LIN {X 0,Y 319.044,Z 405.7,A -85,B 0,C 180,E1 -15783.168,E2 -15783.168} C_VEL
LIN {X 0,Y 320.819,Z 395.688,A -85,B 0,C 180,E1 -15784.719,E2 -15784.719} C_VEL
LIN {X 0,Y 322.608,Z 384.973,A -85,B 0,C 180,E1 -15786.028,E2 -15786.028} C_VEL
LIN {X 0,Y 324.207,Z 372.814,A -85,B 0,C 180,E1 -15787.203,E2 -15787.203} C_VEL
LIN {X 0,Y 325.391,Z 360.596,A -85,B 0,C 180,E1 -15788.09,E2 -15788.09} C_VEL
LIN {X 0,Y 326.349,Z 347.7,A -85,B 0,C 180,E1 -15788.748,E2 -15788.748} C_VEL
LIN {X 0,Y 326.945,Z 334.043,A -85,B 0,C 180,E1 -15789.178,E2 -15789.178} C_VEL
LIN {X 0,Y 329.007,Z 266.698,A -85,B 0,C 180,E1 -15790.66,E2 -15790.66} C_VEL
LIN {X 0,Y 328.282,Z 264.874,A -85,B 0,C 180,E1 -15790.781,E2 -15790.781} C_VEL
LIN {X 0,Y 325.588,Z 260.147,A -85,B 0,C 180,E1 -15791.184,E2 -15791.184} C_VEL
LIN {X 0,Y 319.666,Z 253.624,A -85,B 0,C 180,E1 -15791.999,E2 -15791.999} C_VEL
LIN {X 0,Y 313.621,Z 247.243,A -85,B 0,C 180,E1 -15792.866,E2 -15792.866} C_VEL
LIN {X 0,Y 310.723,Z 242.716,A -85,B 0,C 180,E1 -15793.339,E2 -15793.339} C_VEL
LIN {X 0,Y 306.192,Z 234.216,A -85,B 0,C 180,E1 -15794.15,E2 -15794.15} C_VEL
LIN {X 0,Y 305.555,Z 231.425,A -85,B 0,C 180,E1 -15795.232,E2 -15795.232} C_VEL
LIN {X 0,Y 305.477,Z 231.432,A -85,B 0,C 180,E1 -15799.393,E2 -15799.393} C_VEL
LIN {X 0,Y 305.486,Z 231.431,A -85,B 0,C 180,E1 -15803.263,E2 -15803.263} C_VEL
LIN {X 0,Y 305.453,Z 231.436,A -85,B 0,C 180,E1 -15806.482,E2 -15806.482} C_VEL
LIN {X 0,Y 305.481,Z 231.426,A -85,B 0,C 180,E1 -15810.95,E2 -15810.95} C_VEL
LIN {X 0,Y 305.557,Z 231.416,A -85,B 0,C 180,E1 -15814.087,E2 -15814.087} C_VEL
LIN {X 0,Y 305.488,Z 231.422,A -85,B 0,C 180,E1 -15818.402,E2 -15818.402} C_VEL
LIN {X 0,Y 305.575,Z 231.42,A -85,B 0,C 180,E1 -15821.217,E2 -15821.217} C_VEL
LIN {X 0,Y 305.632,Z 231.416,A -85,B 0,C 180,E1 -15825.349,E2 -15825.349} C_VEL
LIN {X 0,Y 305.616,Z 231.416,A -85,B 0,C 180,E1 -15829.399,E2 -15829.399} C_VEL
LIN {X 0,Y 305.77,Z 231.385,A -85,B 0,C 180,E1 -15832.074,E2 -15832.074} C_VEL
LIN {X 0,Y 305.664,Z 231.407,A -85,B 0,C 180,E1 -15834.723,E2 -15834.723} C_VEL
LIN {X 0,Y 305.935,Z 231.371,A -85,B 0,C 180,E1 -15838.684,E2 -15838.684} C_VEL
LIN {X 0,Y 305.935,Z 231.362,A -85,B 0,C 180,E1 -15841.317,E2 -15841.317} C_VEL
LIN {X 0,Y 305.65,Z 231.397,A -85,B 0,C 180,E1 -15845.278,E2 -15845.278} C_VEL
LIN {X 0,Y 305.734,Z 231.395,A -85,B 0,C 180,E1 -15847.928,E2 -15847.928} C_VEL
LIN {X 0,Y 305.581,Z 231.414,A -85,B 0,C 180,E1 -15851.946,E2 -15851.946} C_VEL
LIN {X 0,Y 305.592,Z 231.407,A -85,B 0,C 180,E1 -15855.013,E2 -15855.013} C_VEL
LIN {X 0,Y 305.497,Z 231.421,A -85,B 0,C 180,E1 -15858.789,E2 -15858.789} C_VEL
LIN {X 0,Y 305.475,Z 231.425,A -85,B 0,C 180,E1 -15863.041,E2 -15863.041} C_VEL
LIN {X 0,Y 305.456,Z 231.435,A -85,B 0,C 180,E1 -15866.197,E2 -15866.197} C_VEL
LIN {X 0,Y 305.435,Z 231.44,A -85,B 0,C 180,E1 -15869.034,E2 -15869.034} C_VEL
LIN {X 0,Y 305.423,Z 231.436,A -85,B 0,C 180,E1 -15871.955,E2 -15871.955} C_VEL
LIN {X 0,Y 305.45,Z 231.434,A -85,B 0,C 180,E1 -15875.115,E2 -15875.115} C_VEL
LIN {X 0,Y 305.426,Z 231.439,A -85,B 0,C 180,E1 -15878.526,E2 -15878.526} C_VEL
LIN {X 0,Y 305.42,Z 231.421,A -85,B 0,C 180,E1 -15881.861,E2 -15881.861} C_VEL
LIN {X 0,Y 305.394,Z 231.441,A -85,B 0,C 180,E1 -15885.513,E2 -15885.513} C_VEL
LIN {X 0,Y 305.407,Z 231.443,A -85,B 0,C 180,E1 -15888.139,E2 -15888.139} C_VEL
LIN {X 0,Y 305.469,Z 231.431,A -85,B 0,C 180,E1 -15892.434,E2 -15892.434} C_VEL
LIN {X 0,Y 305.482,Z 231.57,A -85,B 0,C 180,E1 -15893.005,E2 -15893.005} C_VEL
LIN {X 0,Y 307.845,Z 240.356,A -85,B 0,C 180,E1 -15896.069,E2 -15896.069} C_VEL
LIN {X 0,Y 310.507,Z 251.535,A -85,B 0,C 180,E1 -15899.69,E2 -15899.69} C_VEL
LIN {X 0,Y 311.721,Z 257.855,A -85,B 0,C 180,E1 -15901.611,E2 -15901.611} C_VEL
LIN {X 0,Y 314.185,Z 264.29,A -85,B 0,C 180,E1 -15902.076,E2 -15902.076} C_VEL
LIN {X 0,Y 318.273,Z 283.563,A -85,B 0,C 180,E1 -15903.048,E2 -15903.048} C_VEL
LIN {X 0,Y 321.317,Z 301.733,A -85,B 0,C 180,E1 -15903.846,E2 -15903.846} C_VEL
LIN {X 0,Y 321.763,Z 306.305,A -85,B 0,C 180,E1 -15904.01,E2 -15904.01} C_VEL
LIN {X 0,Y 319.912,Z 367.181,A -85,B 0,C 180,E1 -15905.416,E2 -15905.416} C_VEL
LIN {X 0,Y 318.804,Z 381.015,A -85,B 0,C 180,E1 -15905.975,E2 -15905.975} C_VEL
LIN {X 0,Y 317.356,Z 393.967,A -85,B 0,C 180,E1 -15906.767,E2 -15906.767} C_VEL
LIN {X 0,Y 315.596,Z 405.738,A -85,B 0,C 180,E1 -15907.754,E2 -15907.754} C_VEL
LIN {X 0,Y 313.641,Z 417.083,A -85,B 0,C 180,E1 -15908.99,E2 -15908.99} C_VEL
LIN {X 0,Y 311.742,Z 427.34,A -85,B 0,C 180,E1 -15910.406,E2 -15910.406} C_VEL
LIN {X 0,Y 310.065,Z 435.756,A -85,B 0,C 180,E1 -15911.84,E2 -15911.84} C_VEL
LIN {X 0,Y 308.386,Z 443.923,A -85,B 0,C 180,E1 -15913.539,E2 -15913.539} C_VEL
LIN {X 0,Y 306.93,Z 451.203,A -85,B 0,C 180,E1 -15915.411,E2 -15915.411} C_VEL
LIN {X 0,Y 305.548,Z 457.385,A -85,B 0,C 180,E1 -15917.377,E2 -15917.377} C_VEL
LIN {X 0,Y 304.67,Z 462.324,A -85,B 0,C 180,E1 -15919.364,E2 -15919.364} C_VEL
LIN {X 0,Y 304.061,Z 466.158,A -85,B 0,C 180,E1 -15921.358,E2 -15921.358} C_VEL
LIN {X 0,Y 303.729,Z 468.991,A -85,B 0,C 180,E1 -15923.355,E2 -15923.355} C_VEL
LIN {X 0,Y 303.654,Z 471.313,A -85,B 0,C 180,E1 -15926.017,E2 -15926.017} C_VEL
LIN {X 0,Y 303.655,Z 471.885,A -85,B 0,C 180,E1 -15927.345,E2 -15927.345} C_VEL
LIN {X 0,Y 303.684,Z 472.025,A -85,B 0,C 180,E1 -15928.672,E2 -15928.672} C_VEL
LIN {X 0,Y 303.77,Z 471.772,A -85,B 0,C 180,E1 -15929.998,E2 -15929.998} C_VEL
LIN {X 0,Y 303.724,Z 471.122,A -85,B 0,C 180,E1 -15931.323,E2 -15931.323} C_VEL
LIN {X 0,Y 303.689,Z 470.074,A -85,B 0,C 180,E1 -15932.65,E2 -15932.65} C_VEL
LIN {X 0,Y 303.734,Z 468.569,A -85,B 0,C 180,E1 -15933.978,E2 -15933.978} C_VEL
LIN {X 0,Y 303.73,Z 465.919,A -85,B 0,C 180,E1 -15935.741,E2 -15935.741} C_VEL
LIN {X 0,Y 303.922,Z 461.34,A -85,B 0,C 180,E1 -15937.972,E2 -15937.972} C_VEL
LIN {X 0,Y 304.388,Z 454.961,A -85,B 0,C 180,E1 -15940.305,E2 -15940.305} C_VEL
LIN {X 0,Y 305.056,Z 448,A -85,B 0,C 180,E1 -15942.301,E2 -15942.301} C_VEL
LIN {X 0,Y 305.854,Z 440.881,A -85,B 0,C 180,E1 -15943.958,E2 -15943.958} C_VEL
LIN {X 0,Y 306.85,Z 432.799,A -85,B 0,C 180,E1 -15945.515,E2 -15945.515} C_VEL
LIN {X 0,Y 307.982,Z 422.94,A -85,B 0,C 180,E1 -15947.065,E2 -15947.065} C_VEL
LIN {X 0,Y 309.065,Z 412.504,A -85,B 0,C 180,E1 -15948.388,E2 -15948.388} C_VEL
LIN {X 0,Y 310.317,Z 401.262,A -85,B 0,C 180,E1 -15949.511,E2 -15949.511} C_VEL
LIN {X 0,Y 311.486,Z 388.684,A -85,B 0,C 180,E1 -15950.466,E2 -15950.466} C_VEL
LIN {X 0,Y 312.401,Z 375.211,A -85,B 0,C 180,E1 -15951.179,E2 -15951.179} C_VEL
LIN {X 0,Y 312.939,Z 361.946,A -85,B 0,C 180,E1 -15951.616,E2 -15951.616} C_VEL
LIN {X 0,Y 314.065,Z 301.944,A -85,B 0,C 180,E1 -15952.983,E2 -15952.983} C_VEL
LIN {X 0,Y 308.541,Z 258.947,A -85,B 0,C 180,E1 -15954.397,E2 -15954.397} C_VEL
LIN {X 0,Y 309.359,Z 251.47,A -85,B 0,C 180,E1 -15956.29,E2 -15956.29} C_VEL
LIN {X 0,Y 308.187,Z 244.192,A -85,B 0,C 180,E1 -15958.278,E2 -15958.278} C_VEL
LIN {X 0,Y 305.47,Z 231.437,A -85,B 0,C 180,E1 -15961.943,E2 -15961.943} C_VEL
LIN {X 0,Y 305.447,Z 231.437,A -85,B 0,C 180,E1 -15965.109,E2 -15965.109} C_VEL
LIN {X 0,Y 305.449,Z 231.437,A -85,B 0,C 180,E1 -15968.528,E2 -15968.528} C_VEL
LIN {X 0,Y 305.439,Z 231.436,A -85,B 0,C 180,E1 -15972.582,E2 -15972.582} C_VEL
LIN {X 0,Y 305.464,Z 231.434,A -85,B 0,C 180,E1 -15976.351,E2 -15976.351} C_VEL
LIN {X 0,Y 305.458,Z 231.437,A -85,B 0,C 180,E1 -15979.892,E2 -15979.892} C_VEL
LIN {X 0,Y 305.471,Z 231.435,A -85,B 0,C 180,E1 -15983.623,E2 -15983.623} C_VEL
LIN {X 0,Y 305.435,Z 231.435,A -85,B 0,C 180,E1 -15986.479,E2 -15986.479} C_VEL
LIN {X 0,Y 305.462,Z 231.433,A -85,B 0,C 180,E1 -15990.947,E2 -15990.947} C_VEL
LIN {X 0,Y 305.538,Z 231.424,A -85,B 0,C 180,E1 -15994.084,E2 -15994.084} C_VEL
LIN {X 0,Y 305.474,Z 231.431,A -85,B 0,C 180,E1 -15998.4,E2 -15998.4} C_VEL
LIN {X 0,Y 305.555,Z 231.424,A -85,B 0,C 180,E1 -16001.215,E2 -16001.215} C_VEL
LIN {X 0,Y 305.599,Z 231.42,A -85,B 0,C 180,E1 -16005.346,E2 -16005.346} C_VEL
LIN {X 0,Y 305.599,Z 231.419,A -85,B 0,C 180,E1 -16009.398,E2 -16009.398} C_VEL
LIN {X 0,Y 305.774,Z 231.394,A -85,B 0,C 180,E1 -16012.073,E2 -16012.073} C_VEL
LIN {X 0,Y 305.649,Z 231.41,A -85,B 0,C 180,E1 -16014.722,E2 -16014.722} C_VEL
LIN {X 0,Y 305.914,Z 231.37,A -85,B 0,C 180,E1 -16018.683,E2 -16018.683} C_VEL
LIN {X 0,Y 305.913,Z 231.373,A -85,B 0,C 180,E1 -16021.316,E2 -16021.316} C_VEL
LIN {X 0,Y 305.795,Z 231.393,A -85,B 0,C 180,E1 -16026.598,E2 -16026.598} C_VEL
LIN {X 0,Y 305.659,Z 231.409,A -85,B 0,C 180,E1 -16029.262,E2 -16029.262} C_VEL
LIN {X 0,Y 305.544,Z 231.423,A -85,B 0,C 180,E1 -16033.298,E2 -16033.298} C_VEL
LIN {X 0,Y 305.513,Z 231.426,A -85,B 0,C 180,E1 -16036.024,E2 -16036.024} C_VEL
LIN {X 0,Y 305.442,Z 231.433,A -85,B 0,C 180,E1 -16040.19,E2 -16040.19} C_VEL
LIN {X 0,Y 305.463,Z 231.436,A -85,B 0,C 180,E1 -16044.465,E2 -16044.465} C_VEL
LIN {X 0,Y 305.454,Z 231.43,A -85,B 0,C 180,E1 -16047.397,E2 -16047.397} C_VEL
LIN {X 0,Y 305.4,Z 231.435,A -85,B 0,C 180,E1 -16050.415,E2 -16050.415} C_VEL
LIN {X 0,Y 305.432,Z 231.434,A -85,B 0,C 180,E1 -16054.081,E2 -16054.081} C_VEL
LIN {X 0,Y 305.443,Z 231.437,A -85,B 0,C 180,E1 -16056.743,E2 -16056.743} C_VEL
LIN {X 0,Y 305.426,Z 231.436,A -85,B 0,C 180,E1 -16060.603,E2 -16060.603} C_VEL
LIN {X 0,Y 305.399,Z 231.434,A -85,B 0,C 180,E1 -16063.659,E2 -16063.659} C_VEL
LIN {X 0,Y 305.431,Z 231.436,A -85,B 0,C 180,E1 -16067.419,E2 -16067.419} C_VEL
LIN {X 0,Y 305.446,Z 231.433,A -85,B 0,C 180,E1 -16071.6,E2 -16071.6} C_VEL
LIN {X 0,Y 305.443,Z 231.435,A -85,B 0,C 180,E1 -16074.891,E2 -16074.891} C_VEL
LIN {X 0,Y 305.433,Z 231.437,A -85,B 0,C 180,E1 -16078.36,E2 -16078.36} C_VEL
LIN {X 0,Y 305.498,Z 231.427,A -85,B 0,C 180,E1 -16081.117,E2 -16081.117} C_VEL
LIN {X 0,Y 305.558,Z 231.425,A -85,B 0,C 180,E1 -16084.092,E2 -16084.092} C_VEL
LIN {X 0,Y 305.464,Z 231.434,A -85,B 0,C 180,E1 -16088.405,E2 -16088.405} C_VEL
LIN {X 0,Y 305.509,Z 231.428,A -85,B 0,C 180,E1 -16091.217,E2 -16091.217} C_VEL
LIN {X 0,Y 305.62,Z 231.417,A -85,B 0,C 180,E1 -16095.351,E2 -16095.351} C_VEL
LIN {X 0,Y 305.683,Z 231.491,A -85,B 0,C 180,E1 -16100.053,E2 -16100.053} C_VEL
LIN {X 0,Y 306.015,Z 233.11,A -85,B 0,C 180,E1 -16100.55,E2 -16100.55} C_VEL
LIN {X 0,Y 313.091,Z 253.572,A -85,B 0,C 180,E1 -16101.521,E2 -16101.521} C_VEL
LIN {X 0,Y 314.73,Z 260.384,A -85,B 0,C 180,E1 -16101.791,E2 -16101.791} C_VEL
LIN {X 0,Y 314.373,Z 285.11,A -85,B 0,C 180,E1 -16102.361,E2 -16102.361} C_VEL
LIN {X 0,Y 313.059,Z 340.43,A -85,B 0,C 180,E1 -16103.639,E2 -16103.639} C_VEL
LIN {X 0,Y 312.537,Z 353.529,A -85,B 0,C 180,E1 -16104.195,E2 -16104.195} C_VEL
LIN {X 0,Y 311.713,Z 366.216,A -85,B 0,C 180,E1 -16104.991,E2 -16104.991} C_VEL
LIN {X 0,Y 310.841,Z 377.488,A -85,B 0,C 180,E1 -16105.951,E2 -16105.951} C_VEL
LIN {X 0,Y 309.763,Z 388.459,A -85,B 0,C 180,E1 -16107.153,E2 -16107.153} C_VEL
LIN {X 0,Y 308.537,Z 399.618,A -85,B 0,C 180,E1 -16108.697,E2 -16108.697} C_VEL
LIN {X 0,Y 307.373,Z 409.069,A -85,B 0,C 180,E1 -16110.33,E2 -16110.33} C_VEL
LIN {X 0,Y 306.231,Z 418.169,A -85,B 0,C 180,E1 -16112.304,E2 -16112.304} C_VEL
LIN {X 0,Y 305.336,Z 425.506,A -85,B 0,C 180,E1 -16114.292,E2 -16114.292} C_VEL
LIN {X 0,Y 304.812,Z 430.463,A -85,B 0,C 180,E1 -16115.957,E2 -16115.957} C_VEL
LIN {X 0,Y 304.304,Z 435.287,A -85,B 0,C 180,E1 -16117.967,E2 -16117.967} C_VEL
LIN {X 0,Y 303.921,Z 438.991,A -85,B 0,C 180,E1 -16119.989,E2 -16119.989} C_VEL
LIN {X 0,Y 303.705,Z 441.659,A -85,B 0,C 180,E1 -16122.022,E2 -16122.022} C_VEL
LIN {X 0,Y 303.61,Z 443.031,A -85,B 0,C 180,E1 -16123.538,E2 -16123.538} C_VEL
LIN {X 0,Y 303.57,Z 444.114,A -85,B 0,C 180,E1 -16126.131,E2 -16126.131} C_VEL
LIN {X 0,Y 303.831,Z 443.821,A -85,B 0,C 180,E1 -16128.491,E2 -16128.491} C_VEL
LIN {X 0,Y 304.111,Z 442.765,A -85,B 0,C 180,E1 -16130.283,E2 -16130.283} C_VEL
LIN {X 0,Y 304.84,Z 440.106,A -85,B 0,C 180,E1 -16132.753,E2 -16132.753} C_VEL
LIN {X 0,Y 305.807,Z 436.078,A -85,B 0,C 180,E1 -16135.161,E2 -16135.161} C_VEL
LIN {X 0,Y 306.971,Z 431.245,A -85,B 0,C 180,E1 -16137.251,E2 -16137.251} C_VEL
LIN {X 0,Y 308.396,Z 425.023,A -85,B 0,C 180,E1 -16139.338,E2 -16139.338} C_VEL
LIN {X 0,Y 310.196,Z 417.184,A -85,B 0,C 180,E1 -16141.406,E2 -16141.406} C_VEL
LIN {X 0,Y 312.044,Z 408.279,A -85,B 0,C 180,E1 -16143.26,E2 -16143.26} C_VEL
LIN {X 0,Y 314.028,Z 397.812,A -85,B 0,C 180,E1 -16144.993,E2 -16144.993} C_VEL
LIN {X 0,Y 315.886,Z 387.609,A -85,B 0,C 180,E1 -16146.324,E2 -16146.324} C_VEL
LIN {X 0,Y 317.479,Z 376.292,A -85,B 0,C 180,E1 -16147.498,E2 -16147.498} C_VEL
LIN {X 0,Y 318.893,Z 363.613,A -85,B 0,C 180,E1 -16148.504,E2 -16148.504} C_VEL
LIN {X 0,Y 319.966,Z 351.192,A -85,B 0,C 180,E1 -16149.209,E2 -16149.209} C_VEL
LIN {X 0,Y 320.63,Z 338.269,A -85,B 0,C 180,E1 -16149.685,E2 -16149.685} C_VEL
LIN {X 0,Y 322.785,Z 268.396,A -85,B 0,C 180,E1 -16151.271,E2 -16151.271} C_VEL
LIN {X 0,Y 315.4,Z 251.823,A -85,B 0,C 180,E1 -16152.533,E2 -16152.533} C_VEL
LIN {X 0,Y 310.723,Z 242.716,A -85,B 0,C 180,E1 -16153.339,E2 -16153.339} C_VEL
LIN {X 0,Y 308.62,Z 239.663,A -85,B 0,C 180,E1 -16153.686,E2 -16153.686} C_VEL
LIN {X 0,Y 305.921,Z 237.295,A -85,B 0,C 180,E1 -16154.092,E2 -16154.092} C_VEL
LIN {X 0,Y 302.106,Z 234.95,A -85,B 0,C 180,E1 -16154.708,E2 -16154.708} C_VEL
LIN {X 0,Y 299.721,Z 233.736,A -85,B 0,C 180,E1 -16155.281,E2 -16155.281} C_VEL
LIN {X 0,Y 298.523,Z 232.453,A -85,B 0,C 180,E1 -16155.908,E2 -16155.908} C_VEL
LIN {X 0,Y 298.487,Z 232.313,A -85,B 0,C 180,E1 -16155.971,E2 -16155.971} C_VEL
LIN {X 0,Y 298.445,Z 232.311,A -85,B 0,C 180,E1 -16158.897,E2 -16158.897} C_VEL
LIN {X 0,Y 298.455,Z 232.307,A -85,B 0,C 180,E1 -16163.187,E2 -16163.187} C_VEL
LIN {X 0,Y 298.383,Z 232.315,A -85,B 0,C 180,E1 -16167.199,E2 -16167.199} C_VEL
LIN {X 0,Y 298.419,Z 232.307,A -85,B 0,C 180,E1 -16170.615,E2 -16170.615} C_VEL
LIN {X 0,Y 298.47,Z 232.304,A -85,B 0,C 180,E1 -16173.474,E2 -16173.474} C_VEL
LIN {X 0,Y 298.421,Z 232.309,A -85,B 0,C 180,E1 -16176.698,E2 -16176.698} C_VEL
LIN {X 0,Y 298.527,Z 232.297,A -85,B 0,C 180,E1 -16180.756,E2 -16180.756} C_VEL
LIN {X 0,Y 298.577,Z 232.292,A -85,B 0,C 180,E1 -16184.994,E2 -16184.994} C_VEL
LIN {X 0,Y 298.572,Z 232.291,A -85,B 0,C 180,E1 -16189.146,E2 -16189.146} C_VEL
LIN {X 0,Y 298.715,Z 232.264,A -85,B 0,C 180,E1 -16191.885,E2 -16191.885} C_VEL
LIN {X 0,Y 298.635,Z 232.282,A -85,B 0,C 180,E1 -16194.599,E2 -16194.599} C_VEL
LIN {X 0,Y 298.902,Z 232.247,A -85,B 0,C 180,E1 -16198.653,E2 -16198.653} C_VEL
LIN {X 0,Y 298.902,Z 232.238,A -85,B 0,C 180,E1 -16201.348,E2 -16201.348} C_VEL
LIN {X 0,Y 298.62,Z 232.272,A -85,B 0,C 180,E1 -16205.402,E2 -16205.402} C_VEL
LIN {X 0,Y 298.685,Z 232.273,A -85,B 0,C 180,E1 -16208.116,E2 -16208.116} C_VEL
LIN {X 0,Y 298.533,Z 232.292,A -85,B 0,C 180,E1 -16212.233,E2 -16212.233} C_VEL
LIN {X 0,Y 298.531,Z 232.287,A -85,B 0,C 180,E1 -16215.166,E2 -16215.166} C_VEL
LIN {X 0,Y 298.429,Z 232.302,A -85,B 0,C 180,E1 -16219.618,E2 -16219.618} C_VEL
LIN {X 0,Y 298.408,Z 232.305,A -85,B 0,C 180,E1 -16223.602,E2 -16223.602} C_VEL
LIN {X 0,Y 298.396,Z 232.31,A -85,B 0,C 180,E1 -16226.584,E2 -16226.584} C_VEL
LIN {X 0,Y 298.381,Z 232.317,A -85,B 0,C 180,E1 -16229.646,E2 -16229.646} C_VEL
LIN {X 0,Y 298.381,Z 232.318,A -85,B 0,C 180,E1 -16232.802,E2 -16232.802} C_VEL
LIN {X 0,Y 298.395,Z 232.316,A -85,B 0,C 180,E1 -16236.074,E2 -16236.074} C_VEL
LIN {X 0,Y 298.391,Z 232.317,A -85,B 0,C 180,E1 -16239.49,E2 -16239.49} C_VEL
LIN {X 0,Y 298.395,Z 232.305,A -85,B 0,C 180,E1 -16243.105,E2 -16243.105} C_VEL
LIN {X 0,Y 298.366,Z 232.319,A -85,B 0,C 180,E1 -16246.916,E2 -16246.916} C_VEL
LIN {X 0,Y 298.382,Z 232.312,A -85,B 0,C 180,E1 -16251.012,E2 -16251.012} C_VEL
LIN {X 0,Y 298.437,Z 232.426,A -85,B 0,C 180,E1 -16252.193,E2 -16252.193} C_VEL
LIN {X 0,Y 301.241,Z 242.869,A -85,B 0,C 180,E1 -16255.95,E2 -16255.95} C_VEL
LIN {X 0,Y 303.699,Z 253.234,A -85,B 0,C 180,E1 -16259.396,E2 -16259.396} C_VEL
LIN {X 0,Y 304.566,Z 257.611,A -85,B 0,C 180,E1 -16260.723,E2 -16260.723} C_VEL
LIN {X 0,Y 308.328,Z 266.462,A -85,B 0,C 180,E1 -16261.439,E2 -16261.439} C_VEL
LIN {X 0,Y 311.791,Z 282.576,A -85,B 0,C 180,E1 -16262.292,E2 -16262.292} C_VEL
LIN {X 0,Y 315.043,Z 301.543,A -85,B 0,C 180,E1 -16263.167,E2 -16263.167} C_VEL
LIN {X 0,Y 315.638,Z 307.057,A -85,B 0,C 180,E1 -16263.378,E2 -16263.378} C_VEL
LIN {X 0,Y 313.694,Z 367.539,A -85,B 0,C 180,E1 -16264.807,E2 -16264.807} C_VEL
LIN {X 0,Y 312.542,Z 381.147,A -85,B 0,C 180,E1 -16265.373,E2 -16265.373} C_VEL
LIN {X 0,Y 311.033,Z 393.946,A -85,B 0,C 180,E1 -16266.178,E2 -16266.178} C_VEL
LIN {X 0,Y 309.073,Z 406.434,A -85,B 0,C 180,E1 -16267.259,E2 -16267.259} C_VEL
LIN {X 0,Y 307.058,Z 417.592,A -85,B 0,C 180,E1 -16268.518,E2 -16268.518} C_VEL
LIN {X 0,Y 305.067,Z 427.673,A -85,B 0,C 180,E1 -16269.959,E2 -16269.959} C_VEL
LIN {X 0,Y 302.954,Z 437.601,A -85,B 0,C 180,E1 -16271.749,E2 -16271.749} C_VEL
LIN {X 0,Y 301.077,Z 446.377,A -85,B 0,C 180,E1 -16273.732,E2 -16273.732} C_VEL
LIN {X 0,Y 299.522,Z 453.436,A -85,B 0,C 180,E1 -16275.736,E2 -16275.736} C_VEL
LIN {X 0,Y 298.207,Z 459.105,A -85,B 0,C 180,E1 -16277.753,E2 -16277.753} C_VEL
LIN {X 0,Y 297.415,Z 463.603,A -85,B 0,C 180,E1 -16279.79,E2 -16279.79} C_VEL
LIN {X 0,Y 296.871,Z 467.046,A -85,B 0,C 180,E1 -16281.832,E2 -16281.832} C_VEL
LIN {X 0,Y 296.554,Z 470.103,A -85,B 0,C 180,E1 -16284.559,E2 -16284.559} C_VEL
LIN {X 0,Y 296.568,Z 471.046,A -85,B 0,C 180,E1 -16285.921,E2 -16285.921} C_VEL
LIN {X 0,Y 296.578,Z 471.576,A -85,B 0,C 180,E1 -16287.281,E2 -16287.281} C_VEL
LIN {X 0,Y 296.678,Z 471.407,A -85,B 0,C 180,E1 -16289.998,E2 -16289.998} C_VEL
LIN {X 0,Y 296.634,Z 470.733,A -85,B 0,C 180,E1 -16291.355,E2 -16291.355} C_VEL
LIN {X 0,Y 296.613,Z 469.646,A -85,B 0,C 180,E1 -16292.714,E2 -16292.714} C_VEL
LIN {X 0,Y 296.645,Z 468.102,A -85,B 0,C 180,E1 -16294.073,E2 -16294.073} C_VEL
LIN {X 0,Y 296.649,Z 465.699,A -85,B 0,C 180,E1 -16295.707,E2 -16295.707} C_VEL
LIN {X 0,Y 296.779,Z 462.287,A -85,B 0,C 180,E1 -16297.481,E2 -16297.481} C_VEL
LIN {X 0,Y 297.087,Z 457.291,A -85,B 0,C 180,E1 -16299.528,E2 -16299.528} C_VEL
LIN {X 0,Y 297.619,Z 450.987,A -85,B 0,C 180,E1 -16301.576,E2 -16301.576} C_VEL
LIN {X 0,Y 298.613,Z 443.109,A -85,B 0,C 180,E1 -16303.609,E2 -16303.609} C_VEL
LIN {X 0,Y 299.753,Z 433.712,A -85,B 0,C 180,E1 -16305.545,E2 -16305.545} C_VEL
LIN {X 0,Y 300.879,Z 424.081,A -85,B 0,C 180,E1 -16307.147,E2 -16307.147} C_VEL
LIN {X 0,Y 302.115,Z 412.723,A -85,B 0,C 180,E1 -16308.65,E2 -16308.65} C_VEL
LIN {X 0,Y 303.4,Z 401.611,A -85,B 0,C 180,E1 -16309.798,E2 -16309.798} C_VEL
LIN {X 0,Y 304.599,Z 389.286,A -85,B 0,C 180,E1 -16310.773,E2 -16310.773} C_VEL
LIN {X 0,Y 305.532,Z 376.273,A -85,B 0,C 180,E1 -16311.502,E2 -16311.502} C_VEL
LIN {X 0,Y 306.157,Z 362.407,A -85,B 0,C 180,E1 -16311.987,E2 -16311.987} C_VEL
LIN {X 0,Y 307.265,Z 302.142,A -85,B 0,C 180,E1 -16313.397,E2 -16313.397} C_VEL
LIN {X 0,Y 301.713,Z 258.649,A -85,B 0,C 180,E1 -16314.859,E2 -16314.859} C_VEL
LIN {X 0,Y 302.352,Z 252.052,A -85,B 0,C 180,E1 -16316.575,E2 -16316.575} C_VEL
LIN {X 0,Y 300.485,Z 242.026,A -85,B 0,C 180,E1 -16319.412,E2 -16319.412} C_VEL
LIN {X 0,Y 298.406,Z 232.316,A -85,B 0,C 180,E1 -16322.288,E2 -16322.288} C_VEL
LIN {X 0,Y 298.403,Z 232.318,A -85,B 0,C 180,E1 -16326.065,E2 -16326.065} C_VEL
LIN {X 0,Y 298.391,Z 232.317,A -85,B 0,C 180,E1 -16329.482,E2 -16329.482} C_VEL
LIN {X 0,Y 298.379,Z 232.315,A -85,B 0,C 180,E1 -16333.099,E2 -16333.099} C_VEL
LIN {X 0,Y 298.417,Z 232.31,A -85,B 0,C 180,E1 -16336.923,E2 -16336.923} C_VEL
LIN {X 0,Y 298.401,Z 232.312,A -85,B 0,C 180,E1 -16340.512,E2 -16340.512} C_VEL
LIN {X 0,Y 298.403,Z 232.315,A -85,B 0,C 180,E1 -16343.928,E2 -16343.928} C_VEL
LIN {X 0,Y 298.364,Z 232.319,A -85,B 0,C 180,E1 -16347.98,E2 -16347.98} C_VEL
LIN {X 0,Y 298.43,Z 232.31,A -85,B 0,C 180,E1 -16351.9,E2 -16351.9} C_VEL
LIN {X 0,Y 298.455,Z 232.306,A -85,B 0,C 180,E1 -16354.921,E2 -16354.921} C_VEL
LIN {X 0,Y 298.404,Z 232.314,A -85,B 0,C 180,E1 -16357.862,E2 -16357.862} C_VEL
LIN {X 0,Y 298.521,Z 232.297,A -85,B 0,C 180,E1 -16360.755,E2 -16360.755} C_VEL
LIN {X 0,Y 298.549,Z 232.296,A -85,B 0,C 180,E1 -16364.992,E2 -16364.992} C_VEL
LIN {X 0,Y 298.554,Z 232.294,A -85,B 0,C 180,E1 -16369.145,E2 -16369.145} C_VEL
LIN {X 0,Y 298.72,Z 232.273,A -85,B 0,C 180,E1 -16371.884,E2 -16371.884} C_VEL
LIN {X 0,Y 298.62,Z 232.285,A -85,B 0,C 180,E1 -16374.598,E2 -16374.598} C_VEL
LIN {X 0,Y 298.881,Z 232.245,A -85,B 0,C 180,E1 -16378.652,E2 -16378.652} C_VEL
LIN {X 0,Y 298.88,Z 232.248,A -85,B 0,C 180,E1 -16381.347,E2 -16381.347} C_VEL
LIN {X 0,Y 298.74,Z 232.273,A -85,B 0,C 180,E1 -16386.755,E2 -16386.755} C_VEL
LIN {X 0,Y 298.591,Z 232.288,A -85,B 0,C 180,E1 -16389.483,E2 -16389.483} C_VEL
LIN {X 0,Y 298.504,Z 232.299,A -85,B 0,C 180,E1 -16393.617,E2 -16393.617} C_VEL
LIN {X 0,Y 298.447,Z 232.309,A -85,B 0,C 180,E1 -16396.414,E2 -16396.414} C_VEL
LIN {X 0,Y 298.406,Z 232.308,A -85,B 0,C 180,E1 -16399.619,E2 -16399.619} C_VEL
LIN {X 0,Y 298.392,Z 232.313,A -85,B 0,C 180,E1 -16403.603,E2 -16403.603} C_VEL
LIN {X 0,Y 298.424,Z 232.311,A -85,B 0,C 180,E1 -16406.58,E2 -16406.58} C_VEL
LIN {X 0,Y 298.368,Z 232.307,A -85,B 0,C 180,E1 -16409.646,E2 -16409.646} C_VEL
LIN {X 0,Y 298.36,Z 232.316,A -85,B 0,C 180,E1 -16412.804,E2 -16412.804} C_VEL
LIN {X 0,Y 298.415,Z 232.312,A -85,B 0,C 180,E1 -16416.81,E2 -16416.81} C_VEL
LIN {X 0,Y 298.359,Z 232.313,A -85,B 0,C 180,E1 -16421.091,E2 -16421.091} C_VEL
LIN {X 0,Y 298.374,Z 232.308,A -85,B 0,C 180,E1 -16423.107,E2 -16423.107} C_VEL
LIN {X 0,Y 298.38,Z 232.315,A -85,B 0,C 180,E1 -16426.925,E2 -16426.925} C_VEL
LIN {X 0,Y 298.378,Z 232.312,A -85,B 0,C 180,E1 -16431.012,E2 -16431.012} C_VEL
LIN {X 0,Y 298.399,Z 232.312,A -85,B 0,C 180,E1 -16433.934,E2 -16433.934} C_VEL
LIN {X 0,Y 298.377,Z 232.319,A -85,B 0,C 180,E1 -16437.988,E2 -16437.988} C_VEL
LIN {X 0,Y 298.445,Z 232.31,A -85,B 0,C 180,E1 -16441.908,E2 -16441.908} C_VEL
LIN {X 0,Y 298.471,Z 232.304,A -85,B 0,C 180,E1 -16444.928,E2 -16444.928} C_VEL
LIN {X 0,Y 298.413,Z 232.312,A -85,B 0,C 180,E1 -16449.317,E2 -16449.317} C_VEL
LIN {X 0,Y 298.485,Z 232.307,A -85,B 0,C 180,E1 -16452.18,E2 -16452.18} C_VEL
LIN {X 0,Y 298.579,Z 232.293,A -85,B 0,C 180,E1 -16454.998,E2 -16454.998} C_VEL
LIN {X 0,Y 298.605,Z 232.292,A -85,B 0,C 180,E1 -16459.691,E2 -16459.691} C_VEL
LIN {X 0,Y 298.929,Z 233.618,A -85,B 0,C 180,E1 -16460.061,E2 -16460.061} C_VEL
LIN {X 0,Y 306.528,Z 255.371,A -85,B 0,C 180,E1 -16461.136,E2 -16461.136} C_VEL
LIN {X 0,Y 308.176,Z 262.479,A -85,B 0,C 180,E1 -16461.42,E2 -16461.42} C_VEL
LIN {X 0,Y 306.282,Z 340.747,A -85,B 0,C 180,E1 -16463.251,E2 -16463.251} C_VEL
LIN {X 0,Y 305.741,Z 353.817,A -85,B 0,C 180,E1 -16463.817,E2 -16463.817} C_VEL
LIN {X 0,Y 304.892,Z 366.516,A -85,B 0,C 180,E1 -16464.63,E2 -16464.63} C_VEL
LIN {X 0,Y 303.915,Z 378.591,A -85,B 0,C 180,E1 -16465.693,E2 -16465.693} C_VEL
LIN {X 0,Y 302.805,Z 389.648,A -85,B 0,C 180,E1 -16466.952,E2 -16466.952} C_VEL
LIN {X 0,Y 301.541,Z 400.472,A -85,B 0,C 180,E1 -16468.5,E2 -16468.5} C_VEL
LIN {X 0,Y 300.461,Z 408.962,A -85,B 0,C 180,E1 -16470.002,E2 -16470.002} C_VEL
LIN {X 0,Y 299.266,Z 418.149,A -85,B 0,C 180,E1 -16472.021,E2 -16472.021} C_VEL
LIN {X 0,Y 298.335,Z 425.545,A -85,B 0,C 180,E1 -16474.055,E2 -16474.055} C_VEL
LIN {X 0,Y 297.697,Z 431.47,A -85,B 0,C 180,E1 -16476.1,E2 -16476.1} C_VEL
LIN {X 0,Y 297.159,Z 436.156,A -85,B 0,C 180,E1 -16478.16,E2 -16478.16} C_VEL
LIN {X 0,Y 296.798,Z 439.726,A -85,B 0,C 180,E1 -16480.231,E2 -16480.231} C_VEL
LIN {X 0,Y 296.581,Z 442.27,A -85,B 0,C 180,E1 -16482.315,E2 -16482.315} C_VEL
LIN {X 0,Y 296.512,Z 443.423,A -85,B 0,C 180,E1 -16483.712,E2 -16483.712} C_VEL
LIN {X 0,Y 296.44,Z 444.152,A -85,B 0,C 180,E1 -16485.118,E2 -16485.118} C_VEL
LIN {X 0,Y 296.497,Z 444.48,A -85,B 0,C 180,E1 -16486.526,E2 -16486.526} C_VEL
LIN {X 0,Y 296.772,Z 444.148,A -85,B 0,C 180,E1 -16488.692,E2 -16488.692} C_VEL
LIN {X 0,Y 297.146,Z 442.884,A -85,B 0,C 180,E1 -16490.78,E2 -16490.78} C_VEL
LIN {X 0,Y 297.877,Z 440.423,A -85,B 0,C 180,E1 -16493.053,E2 -16493.053} C_VEL
LIN {X 0,Y 298.67,Z 437.241,A -85,B 0,C 180,E1 -16495.059,E2 -16495.059} C_VEL
LIN {X 0,Y 299.914,Z 432.43,A -85,B 0,C 180,E1 -16497.312,E2 -16497.312} C_VEL
LIN {X 0,Y 301.587,Z 425.666,A -85,B 0,C 180,E1 -16499.682,E2 -16499.682} C_VEL
LIN {X 0,Y 303.451,Z 417.893,A -85,B 0,C 180,E1 -16501.795,E2 -16501.795} C_VEL
LIN {X 0,Y 305.227,Z 409.852,A -85,B 0,C 180,E1 -16503.546,E2 -16503.546} C_VEL
LIN {X 0,Y 307.271,Z 399.877,A -85,B 0,C 180,E1 -16505.276,E2 -16505.276} C_VEL
LIN {X 0,Y 309.386,Z 388.762,A -85,B 0,C 180,E1 -16506.796,E2 -16506.796} C_VEL
LIN {X 0,Y 311.048,Z 377.617,A -85,B 0,C 180,E1 -16508.002,E2 -16508.002} C_VEL
LIN {X 0,Y 312.514,Z 365.227,A -85,B 0,C 180,E1 -16509.025,E2 -16509.025} C_VEL
LIN {X 0,Y 313.664,Z 352.5,A -85,B 0,C 180,E1 -16509.788,E2 -16509.788} C_VEL
LIN {X 0,Y 314.372,Z 340.811,A -85,B 0,C 180,E1 -16510.255,E2 -16510.255} C_VEL
LIN {X 0,Y 316.741,Z 270.516,A -85,B 0,C 180,E1 -16511.879,E2 -16511.879} C_VEL
LIN {X 0,Y 310.055,Z 255.508,A -85,B 0,C 180,E1 -16513.068,E2 -16513.068} C_VEL
LIN {X 0,Y 302.281,Z 240.681,A -85,B 0,C 180,E1 -16514.467,E2 -16514.467} C_VEL
LIN {X 0,Y 299.104,Z 234.571,A -85,B 0,C 180,E1 -16515.092,E2 -16515.092} C_VEL
LIN {X 0,Y 298.487,Z 232.313,A -85,B 0,C 180,E1 -16515.971,E2 -16515.971} C_VEL
LIN {X 0,Y 297.915,Z 232.378,A -85,B 0,C 180,E1 -16516.704,E2 -16516.704} C_VEL
LIN {X 0,Y 295.823,Z 232.635,A -85,B 0,C 180,E1 -16518.172,E2 -16518.172} C_VEL
LIN {X 0,Y 292.343,Z 233.199,A -85,B 0,C 180,E1 -16520.405,E2 -16520.405} C_VEL
LIN {X 0,Y 291.418,Z 233.195,A -85,B 0,C 180,E1 -16521.567,E2 -16521.567} C_VEL
LIN {X 0,Y 291.351,Z 233.188,A -85,B 0,C 180,E1 -16521.96,E2 -16521.96} C_VEL
LIN {X 0,Y 291.362,Z 233.184,A -85,B 0,C 180,E1 -16525.093,E2 -16525.093} C_VEL
LIN {X 0,Y 291.359,Z 233.184,A -85,B 0,C 180,E1 -16527.95,E2 -16527.95} C_VEL
LIN {X 0,Y 291.369,Z 233.182,A -85,B 0,C 180,E1 -16531.157,E2 -16531.157} C_VEL
LIN {X 0,Y 291.403,Z 233.178,A -85,B 0,C 180,E1 -16534.271,E2 -16534.271} C_VEL
LIN {X 0,Y 291.368,Z 233.189,A -85,B 0,C 180,E1 -16537.299,E2 -16537.299} C_VEL
LIN {X 0,Y 291.447,Z 233.178,A -85,B 0,C 180,E1 -16540.27,E2 -16540.27} C_VEL
LIN {X 0,Y 291.527,Z 233.169,A -85,B 0,C 180,E1 -16544.634,E2 -16544.634} C_VEL
LIN {X 0,Y 291.517,Z 233.169,A -85,B 0,C 180,E1 -16548.88,E2 -16548.88} C_VEL
LIN {X 0,Y 291.663,Z 233.142,A -85,B 0,C 180,E1 -16551.688,E2 -16551.688} C_VEL
LIN {X 0,Y 291.606,Z 233.158,A -85,B 0,C 180,E1 -16554.468,E2 -16554.468} C_VEL
LIN {X 0,Y 291.869,Z 233.123,A -85,B 0,C 180,E1 -16558.621,E2 -16558.621} C_VEL
LIN {X 0,Y 291.868,Z 233.113,A -85,B 0,C 180,E1 -16561.38,E2 -16561.38} C_VEL
LIN {X 0,Y 291.675,Z 233.141,A -85,B 0,C 180,E1 -16566.92,E2 -16566.92} C_VEL
LIN {X 0,Y 291.553,Z 233.153,A -85,B 0,C 180,E1 -16569.715,E2 -16569.715} C_VEL
LIN {X 0,Y 291.499,Z 233.165,A -85,B 0,C 180,E1 -16573.952,E2 -16573.952} C_VEL
LIN {X 0,Y 291.409,Z 233.184,A -85,B 0,C 180,E1 -16576.823,E2 -16576.823} C_VEL
LIN {X 0,Y 291.379,Z 233.181,A -85,B 0,C 180,E1 -16579.843,E2 -16579.843} C_VEL
LIN {X 0,Y 291.347,Z 233.187,A -85,B 0,C 180,E1 -16584.21,E2 -16584.21} C_VEL
LIN {X 0,Y 291.342,Z 233.186,A -85,B 0,C 180,E1 -16587.28,E2 -16587.28} C_VEL
LIN {X 0,Y 291.305,Z 233.194,A -85,B 0,C 180,E1 -16590.441,E2 -16590.441} C_VEL
LIN {X 0,Y 291.333,Z 233.193,A -85,B 0,C 180,E1 -16593.7,E2 -16593.7} C_VEL
LIN {X 0,Y 291.35,Z 233.188,A -85,B 0,C 180,E1 -16597.25,E2 -16597.25} C_VEL
LIN {X 0,Y 291.321,Z 233.184,A -85,B 0,C 180,E1 -16600.645,E2 -16600.645} C_VEL
LIN {X 0,Y 291.287,Z 233.203,A -85,B 0,C 180,E1 -16604.403,E2 -16604.403} C_VEL
LIN {X 0,Y 291.291,Z 233.203,A -85,B 0,C 180,E1 -16608.413,E2 -16608.413} C_VEL
LIN {X 0,Y 291.375,Z 233.266,A -85,B 0,C 180,E1 -16611.321,E2 -16611.321} C_VEL
LIN {X 0,Y 294.082,Z 243.056,A -85,B 0,C 180,E1 -16615.002,E2 -16615.002} C_VEL
LIN {X 0,Y 296.726,Z 254.326,A -85,B 0,C 180,E1 -16618.883,E2 -16618.883} C_VEL
LIN {X 0,Y 297.315,Z 257.08,A -85,B 0,C 180,E1 -16619.762,E2 -16619.762} C_VEL
LIN {X 0,Y 302.874,Z 269.89,A -85,B 0,C 180,E1 -16620.858,E2 -16620.858} C_VEL
LIN {X 0,Y 306.633,Z 288.345,A -85,B 0,C 180,E1 -16621.84,E2 -16621.84} C_VEL
LIN {X 0,Y 309.503,Z 306.524,A -85,B 0,C 180,E1 -16622.676,E2 -16622.676} C_VEL
LIN {X 0,Y 307.63,Z 366.522,A -85,B 0,C 180,E1 -16624.127,E2 -16624.127} C_VEL
LIN {X 0,Y 306.466,Z 379.782,A -85,B 0,C 180,E1 -16624.67,E2 -16624.67} C_VEL
LIN {X 0,Y 304.903,Z 392.9,A -85,B 0,C 180,E1 -16625.487,E2 -16625.487} C_VEL
LIN {X 0,Y 303.174,Z 403.982,A -85,B 0,C 180,E1 -16626.429,E2 -16626.429} C_VEL
LIN {X 0,Y 300.944,Z 415.535,A -85,B 0,C 180,E1 -16627.698,E2 -16627.698} C_VEL
LIN {X 0,Y 298.881,Z 425.942,A -85,B 0,C 180,E1 -16629.166,E2 -16629.166} C_VEL
LIN {X 0,Y 296.967,Z 434.48,A -85,B 0,C 180,E1 -16630.65,E2 -16630.65} C_VEL
LIN {X 0,Y 295.053,Z 443.131,A -85,B 0,C 180,E1 -16632.507,E2 -16632.507} C_VEL
LIN {X 0,Y 293.173,Z 451.26,A -85,B 0,C 180,E1 -16634.71,E2 -16634.71} C_VEL
LIN {X 0,Y 291.664,Z 457.303,A -85,B 0,C 180,E1 -16636.766,E2 -16636.766} C_VEL
LIN {X 0,Y 290.666,Z 462.114,A -85,B 0,C 180,E1 -16638.845,E2 -16638.845} C_VEL
LIN {X 0,Y 289.993,Z 465.833,A -85,B 0,C 180,E1 -16640.935,E2 -16640.935} C_VEL
LIN {X 0,Y 289.58,Z 468.557,A -85,B 0,C 180,E1 -16643.028,E2 -16643.028} C_VEL
LIN {X 0,Y 289.483,Z 469.924,A -85,B 0,C 180,E1 -16644.5,E2 -16644.5} C_VEL
LIN {X 0,Y 289.465,Z 470.776,A -85,B 0,C 180,E1 -16645.821,E2 -16645.821} C_VEL
LIN {X 0,Y 289.503,Z 471.26,A -85,B 0,C 180,E1 -16647.215,E2 -16647.215} C_VEL
LIN {X 0,Y 289.588,Z 471.042,A -85,B 0,C 180,E1 -16649.998,E2 -16649.998} C_VEL
LIN {X 0,Y 289.548,Z 470.344,A -85,B 0,C 180,E1 -16651.388,E2 -16651.388} C_VEL
LIN {X 0,Y 289.539,Z 469.207,A -85,B 0,C 180,E1 -16652.78,E2 -16652.78} C_VEL
LIN {X 0,Y 289.532,Z 466.345,A -85,B 0,C 180,E1 -16655.108,E2 -16655.108} C_VEL
LIN {X 0,Y 289.705,Z 461.736,A -85,B 0,C 180,E1 -16657.664,E2 -16657.664} C_VEL
LIN {X 0,Y 290.053,Z 456.68,A -85,B 0,C 180,E1 -16659.762,E2 -16659.762} C_VEL
LIN {X 0,Y 290.634,Z 450.306,A -85,B 0,C 180,E1 -16661.858,E2 -16661.858} C_VEL
LIN {X 0,Y 291.628,Z 442.306,A -85,B 0,C 180,E1 -16663.941,E2 -16663.941} C_VEL
LIN {X 0,Y 292.776,Z 433.325,A -85,B 0,C 180,E1 -16665.824,E2 -16665.824} C_VEL
LIN {X 0,Y 294.057,Z 423.048,A -85,B 0,C 180,E1 -16667.558,E2 -16667.558} C_VEL
LIN {X 0,Y 295.171,Z 412.913,A -85,B 0,C 180,E1 -16668.926,E2 -16668.926} C_VEL
LIN {X 0,Y 296.492,Z 401.921,A -85,B 0,C 180,E1 -16670.098,E2 -16670.098} C_VEL
LIN {X 0,Y 297.72,Z 389.766,A -85,B 0,C 180,E1 -16671.095,E2 -16671.095} C_VEL
LIN {X 0,Y 298.645,Z 377.222,A -85,B 0,C 180,E1 -16671.841,E2 -16671.841} C_VEL
LIN {X 0,Y 299.299,Z 364.948,A -85,B 0,C 180,E1 -16672.312,E2 -16672.312} C_VEL
LIN {X 0,Y 300.626,Z 303.521,A -85,B 0,C 180,E1 -16673.784,E2 -16673.784} C_VEL
LIN {X 0,Y 294.869,Z 258.279,A -85,B 0,C 180,E1 -16675.357,E2 -16675.357} C_VEL
LIN {X 0,Y 295.328,Z 252.606,A -85,B 0,C 180,E1 -16676.876,E2 -16676.876} C_VEL
LIN {X 0,Y 293.051,Z 240.865,A -85,B 0,C 180,E1 -16680.303,E2 -16680.303} C_VEL
LIN {X 0,Y 291.357,Z 233.193,A -85,B 0,C 180,E1 -16682.679,E2 -16682.679} C_VEL
LIN {X 0,Y 291.394,Z 233.188,A -85,B 0,C 180,E1 -16687.075,E2 -16687.075} C_VEL
LIN {X 0,Y 291.316,Z 233.196,A -85,B 0,C 180,E1 -16690.638,E2 -16690.638} C_VEL
LIN {X 0,Y 291.294,Z 233.198,A -85,B 0,C 180,E1 -16694.393,E2 -16694.393} C_VEL
LIN {X 0,Y 291.357,Z 233.191,A -85,B 0,C 180,E1 -16698.388,E2 -16698.388} C_VEL
LIN {X 0,Y 291.352,Z 233.191,A -85,B 0,C 180,E1 -16701.158,E2 -16701.158} C_VEL
LIN {X 0,Y 291.34,Z 233.192,A -85,B 0,C 180,E1 -16704.623,E2 -16704.623} C_VEL
LIN {X 0,Y 291.341,Z 233.194,A -85,B 0,C 180,E1 -16707.946,E2 -16707.946} C_VEL
LIN {X 0,Y 291.35,Z 233.191,A -85,B 0,C 180,E1 -16711.154,E2 -16711.154} C_VEL
LIN {X 0,Y 291.385,Z 233.186,A -85,B 0,C 180,E1 -16714.268,E2 -16714.268} C_VEL
LIN {X 0,Y 291.372,Z 233.19,A -85,B 0,C 180,E1 -16717.298,E2 -16717.298} C_VEL
LIN {X 0,Y 291.47,Z 233.175,A -85,B 0,C 180,E1 -16720.271,E2 -16720.271} C_VEL
LIN {X 0,Y 291.48,Z 233.175,A -85,B 0,C 180,E1 -16724.65,E2 -16724.65} C_VEL
LIN {X 0,Y 291.498,Z 233.171,A -85,B 0,C 180,E1 -16728.879,E2 -16728.879} C_VEL
LIN {X 0,Y 291.671,Z 233.152,A -85,B 0,C 180,E1 -16731.687,E2 -16731.687} C_VEL
LIN {X 0,Y 291.591,Z 233.159,A -85,B 0,C 180,E1 -16734.467,E2 -16734.467} C_VEL
LIN {X 0,Y 291.847,Z 233.119,A -85,B 0,C 180,E1 -16738.62,E2 -16738.62} C_VEL
LIN {X 0,Y 291.846,Z 233.123,A -85,B 0,C 180,E1 -16741.379,E2 -16741.379} C_VEL
LIN {X 0,Y 291.688,Z 233.153,A -85,B 0,C 180,E1 -16746.919,E2 -16746.919} C_VEL
LIN {X 0,Y 291.533,Z 233.166,A -85,B 0,C 180,E1 -16749.715,E2 -16749.715} C_VEL
LIN {X 0,Y 291.475,Z 233.174,A -85,B 0,C 180,E1 -16753.952,E2 -16753.952} C_VEL
LIN {X 0,Y 291.392,Z 233.189,A -85,B 0,C 180,E1 -16756.823,E2 -16756.823} C_VEL
LIN {X 0,Y 291.355,Z 233.186,A -85,B 0,C 180,E1 -16759.844,E2 -16759.844} C_VEL
LIN {X 0,Y 291.342,Z 233.193,A -85,B 0,C 180,E1 -16764.21,E2 -16764.21} C_VEL
LIN {X 0,Y 291.367,Z 233.184,A -85,B 0,C 180,E1 -16767.277,E2 -16767.277} C_VEL
LIN {X 0,Y 291.288,Z 233.188,A -85,B 0,C 180,E1 -16770.442,E2 -16770.442} C_VEL
LIN {X 0,Y 291.311,Z 233.19,A -85,B 0,C 180,E1 -16773.702,E2 -16773.702} C_VEL
LIN {X 0,Y 291.345,Z 233.191,A -85,B 0,C 180,E1 -16777.257,E2 -16777.257} C_VEL
LIN {X 0,Y 291.304,Z 233.193,A -85,B 0,C 180,E1 -16780.647,E2 -16780.647} C_VEL
LIN {X 0,Y 291.266,Z 233.198,A -85,B 0,C 180,E1 -16784.406,E2 -16784.406} C_VEL
LIN {X 0,Y 291.303,Z 233.2,A -85,B 0,C 180,E1 -16788.409,E2 -16788.409} C_VEL
LIN {X 0,Y 291.327,Z 233.19,A -85,B 0,C 180,E1 -16791.161,E2 -16791.161} C_VEL
LIN {X 0,Y 291.343,Z 233.193,A -85,B 0,C 180,E1 -16794.63,E2 -16794.63} C_VEL
LIN {X 0,Y 291.354,Z 233.194,A -85,B 0,C 180,E1 -16797.955,E2 -16797.955} C_VEL
LIN {X 0,Y 291.363,Z 233.188,A -85,B 0,C 180,E1 -16801.162,E2 -16801.162} C_VEL
LIN {X 0,Y 291.401,Z 233.187,A -85,B 0,C 180,E1 -16804.276,E2 -16804.276} C_VEL
LIN {X 0,Y 291.362,Z 233.19,A -85,B 0,C 180,E1 -16807.303,E2 -16807.303} C_VEL
LIN {X 0,Y 291.397,Z 233.188,A -85,B 0,C 180,E1 -16810.27,E2 -16810.27} C_VEL
LIN {X 0,Y 291.491,Z 233.177,A -85,B 0,C 180,E1 -16814.669,E2 -16814.669} C_VEL
LIN {X 0,Y 291.571,Z 233.168,A -85,B 0,C 180,E1 -16819.202,E2 -16819.202} C_VEL
LIN {X 0,Y 291.618,Z 233.549,A -85,B 0,C 180,E1 -16819.466,E2 -16819.466} C_VEL
LIN {X 0,Y 292.652,Z 236.348,A -85,B 0,C 180,E1 -16819.67,E2 -16819.67} C_VEL
LIN {X 0,Y 299.992,Z 257.231,A -85,B 0,C 180,E1 -16820.738,E2 -16820.738} C_VEL
LIN {X 0,Y 301.423,Z 262.933,A -85,B 0,C 180,E1 -16820.98,E2 -16820.98} C_VEL
LIN {X 0,Y 299.505,Z 341.307,A -85,B 0,C 180,E1 -16822.86,E2 -16822.86} C_VEL
LIN {X 0,Y 298.913,Z 354.766,A -85,B 0,C 180,E1 -16823.464,E2 -16823.464} C_VEL
LIN {X 0,Y 298.084,Z 366.739,A -85,B 0,C 180,E1 -16824.252,E2 -16824.252} C_VEL
LIN {X 0,Y 297.152,Z 378.046,A -85,B 0,C 180,E1 -16825.254,E2 -16825.254} C_VEL
LIN {X 0,Y 295.995,Z 389.331,A -85,B 0,C 180,E1 -16826.549,E2 -16826.549} C_VEL
LIN {X 0,Y 294.678,Z 400.217,A -85,B 0,C 180,E1 -16828.123,E2 -16828.123} C_VEL
LIN {X 0,Y 293.574,Z 408.802,A -85,B 0,C 180,E1 -16829.659,E2 -16829.659} C_VEL
LIN {X 0,Y 292.481,Z 416.726,A -85,B 0,C 180,E1 -16831.379,E2 -16831.379} C_VEL
LIN {X 0,Y 291.492,Z 424.444,A -85,B 0,C 180,E1 -16833.458,E2 -16833.458} C_VEL
LIN {X 0,Y 290.714,Z 430.646,A -85,B 0,C 180,E1 -16835.551,E2 -16835.551} C_VEL
LIN {X 0,Y 290.194,Z 435.564,A -85,B 0,C 180,E1 -16837.656,E2 -16837.656} C_VEL
LIN {X 0,Y 289.776,Z 439.364,A -85,B 0,C 180,E1 -16839.776,E2 -16839.776} C_VEL
LIN {X 0,Y 289.56,Z 441.331,A -85,B 0,C 180,E1 -16841.198,E2 -16841.198} C_VEL
LIN {X 0,Y 289.425,Z 443.734,A -85,B 0,C 180,E1 -16843.761,E2 -16843.761} C_VEL
LIN {X 0,Y 289.349,Z 444.578,A -85,B 0,C 180,E1 -16845.498,E2 -16845.498} C_VEL
LIN {X 0,Y 289.441,Z 444.841,A -85,B 0,C 180,E1 -16846.941,E2 -16846.941} C_VEL
LIN {X 0,Y 289.733,Z 444.472,A -85,B 0,C 180,E1 -16848.914,E2 -16848.914} C_VEL
LIN {X 0,Y 290.197,Z 443.007,A -85,B 0,C 180,E1 -16851.302,E2 -16851.302} C_VEL
LIN {X 0,Y 290.91,Z 440.756,A -85,B 0,C 180,E1 -16853.361,E2 -16853.361} C_VEL
LIN {X 0,Y 291.879,Z 437.104,A -85,B 0,C 180,E1 -16855.684,E2 -16855.684} C_VEL
LIN {X 0,Y 293.206,Z 432.312,A -85,B 0,C 180,E1 -16857.904,E2 -16857.904} C_VEL
LIN {X 0,Y 294.763,Z 426.307,A -85,B 0,C 180,E1 -16860.046,E2 -16860.046} C_VEL
LIN {X 0,Y 296.717,Z 418.602,A -85,B 0,C 180,E1 -16862.203,E2 -16862.203} C_VEL
LIN {X 0,Y 298.58,Z 410.643,A -85,B 0,C 180,E1 -16863.988,E2 -16863.988} C_VEL
LIN {X 0,Y 300.709,Z 400.81,A -85,B 0,C 180,E1 -16865.752,E2 -16865.752} C_VEL
LIN {X 0,Y 302.674,Z 391.11,A -85,B 0,C 180,E1 -16867.135,E2 -16867.135} C_VEL
LIN {X 0,Y 304.42,Z 380.282,A -85,B 0,C 180,E1 -16868.387,E2 -16868.387} C_VEL
LIN {X 0,Y 306.067,Z 368.085,A -85,B 0,C 180,E1 -16869.476,E2 -16869.476} C_VEL
LIN {X 0,Y 307.328,Z 355.459,A -85,B 0,C 180,E1 -16870.295,E2 -16870.295} C_VEL
LIN {X 0,Y 308.176,Z 342.693,A -85,B 0,C 180,E1 -16870.859,E2 -16870.859} C_VEL
LIN {X 0,Y 309.974,Z 293.201,A -85,B 0,C 180,E1 -16872.046,E2 -16872.046} C_VEL
LIN {X 0,Y 310.56,Z 272.286,A -85,B 0,C 180,E1 -16872.547,E2 -16872.547} C_VEL
LIN {X 0,Y 304.558,Z 258.834,A -85,B 0,C 180,E1 -16873.655,E2 -16873.655} C_VEL
LIN {X 0,Y 297.456,Z 245.139,A -85,B 0,C 180,E1 -16874.982,E2 -16874.982} C_VEL
LIN {X 0,Y 293.243,Z 237.697,A -85,B 0,C 180,E1 -16875.792,E2 -16875.792} C_VEL
LIN {X 0,Y 291.9,Z 234.984,A -85,B 0,C 180,E1 -16876.092,E2 -16876.092} C_VEL
LIN {X 0,Y 291.445,Z 233.182,A -85,B 0,C 180,E1 -16876.88,E2 -16876.88} C_VEL
LIN {X 0,Y 291.369,Z 233.192,A -85,B 0,C 180,E1 -16881.161,E2 -16881.161} C_VEL
LIN {X 0,Y 291.351,Z 233.188,A -85,B 0,C 180,E1 -16881.96,E2 -16881.96} C_VEL
LIN {X 0,Y 290.694,Z 233.273,A -85,B 0,C 180,E1 -16883.113,E2 -16883.113} C_VEL
LIN {X 0,Y 287.825,Z 233.626,A -85,B 0,C 180,E1 -16884.99,E2 -16884.99} C_VEL
LIN {X 0,Y 285.386,Z 233.936,A -85,B 0,C 180,E1 -16886.514,E2 -16886.514} C_VEL
LIN {X 0,Y 284.345,Z 234.059,A -85,B 0,C 180,E1 -16887.696,E2 -16887.696} C_VEL
LIN {X 0,Y 284.264,Z 234.067,A -85,B 0,C 180,E1 -16888.096,E2 -16888.096} C_VEL
LIN {X 0,Y 284.346,Z 234.061,A -85,B 0,C 180,E1 -16890.375,E2 -16890.375} C_VEL
LIN {X 0,Y 284.366,Z 234.061,A -85,B 0,C 180,E1 -16893.586,E2 -16893.586} C_VEL
LIN {X 0,Y 284.353,Z 234.061,A -85,B 0,C 180,E1 -16896.706,E2 -16896.706} C_VEL
LIN {X 0,Y 284.391,Z 234.06,A -85,B 0,C 180,E1 -16901.261,E2 -16901.261} C_VEL
LIN {X 0,Y 284.465,Z 234.049,A -85,B 0,C 180,E1 -16904.47,E2 -16904.47} C_VEL
LIN {X 0,Y 284.469,Z 234.046,A -85,B 0,C 180,E1 -16908.601,E2 -16908.601} C_VEL
LIN {X 0,Y 284.616,Z 234.021,A -85,B 0,C 180,E1 -16911.48,E2 -16911.48} C_VEL
LIN {X 0,Y 284.576,Z 234.033,A -85,B 0,C 180,E1 -16914.331,E2 -16914.331} C_VEL
LIN {X 0,Y 284.835,Z 233.999,A -85,B 0,C 180,E1 -16918.587,E2 -16918.587} C_VEL
LIN {X 0,Y 284.835,Z 233.989,A -85,B 0,C 180,E1 -16921.414,E2 -16921.414} C_VEL
LIN {X 0,Y 284.63,Z 234.02,A -85,B 0,C 180,E1 -16927.092,E2 -16927.092} C_VEL
LIN {X 0,Y 284.499,Z 234.03,A -85,B 0,C 180,E1 -16929.958,E2 -16929.958} C_VEL
LIN {X 0,Y 284.448,Z 234.041,A -85,B 0,C 180,E1 -16934.305,E2 -16934.305} C_VEL
LIN {X 0,Y 284.313,Z 234.059,A -85,B 0,C 180,E1 -16938.745,E2 -16938.745} C_VEL
LIN {X 0,Y 284.315,Z 234.06,A -85,B 0,C 180,E1 -16943.298,E2 -16943.298} C_VEL
LIN {X 0,Y 284.318,Z 234.06,A -85,B 0,C 180,E1 -16947.147,E2 -16947.147} C_VEL
LIN {X 0,Y 284.284,Z 234.071,A -85,B 0,C 180,E1 -16950.092,E2 -16950.092} C_VEL
LIN {X 0,Y 284.276,Z 234.075,A -85,B 0,C 180,E1 -16952.95,E2 -16952.95} C_VEL
LIN {X 0,Y 284.312,Z 234.071,A -85,B 0,C 180,E1 -16956.389,E2 -16956.389} C_VEL
LIN {X 0,Y 284.3,Z 234.066,A -85,B 0,C 180,E1 -16959.996,E2 -16959.996} C_VEL
LIN {X 0,Y 284.243,Z 234.081,A -85,B 0,C 180,E1 -16964.192,E2 -16964.192} C_VEL
LIN {X 0,Y 284.236,Z 234.08,A -85,B 0,C 180,E1 -16968.119,E2 -16968.119} C_VEL
LIN {X 0,Y 284.328,Z 234.197,A -85,B 0,C 180,E1 -16970.427,E2 -16970.427} C_VEL
LIN {X 0,Y 286.845,Z 243.26,A -85,B 0,C 180,E1 -16973.984,E2 -16973.984} C_VEL
LIN {X 0,Y 289.073,Z 252.27,A -85,B 0,C 180,E1 -16977.252,E2 -16977.252} C_VEL
LIN {X 0,Y 290.11,Z 256.803,A -85,B 0,C 180,E1 -16978.752,E2 -16978.752} C_VEL
LIN {X 0,Y 297.172,Z 272.198,A -85,B 0,C 180,E1 -16980.186,E2 -16980.186} C_VEL
LIN {X 0,Y 300.766,Z 290.21,A -85,B 0,C 180,E1 -16981.171,E2 -16981.171} C_VEL
LIN {X 0,Y 303.408,Z 306.943,A -85,B 0,C 180,E1 -16981.968,E2 -16981.968} C_VEL
LIN {X 0,Y 303.209,Z 317.768,A -85,B 0,C 180,E1 -16982.246,E2 -16982.246} C_VEL
LIN {X 0,Y 301.495,Z 366.922,A -85,B 0,C 180,E1 -16983.461,E2 -16983.461} C_VEL
LIN {X 0,Y 300.217,Z 380.78,A -85,B 0,C 180,E1 -16984.058,E2 -16984.058} C_VEL
LIN {X 0,Y 298.662,Z 392.968,A -85,B 0,C 180,E1 -16984.847,E2 -16984.847} C_VEL
LIN {X 0,Y 296.722,Z 404.728,A -85,B 0,C 180,E1 -16985.884,E2 -16985.884} C_VEL
LIN {X 0,Y 294.423,Z 416.076,A -85,B 0,C 180,E1 -16987.176,E2 -16987.176} C_VEL
LIN {X 0,Y 292.275,Z 426.326,A -85,B 0,C 180,E1 -16988.672,E2 -16988.672} C_VEL
LIN {X 0,Y 289.892,Z 436.382,A -85,B 0,C 180,E1 -16990.527,E2 -16990.527} C_VEL
LIN {X 0,Y 287.808,Z 445.15,A -85,B 0,C 180,E1 -16992.568,E2 -16992.568} C_VEL
LIN {X 0,Y 286.048,Z 452.41,A -85,B 0,C 180,E1 -16994.684,E2 -16994.684} C_VEL
LIN {X 0,Y 284.283,Z 458.971,A -85,B 0,C 180,E1 -16997.143,E2 -16997.143} C_VEL
LIN {X 0,Y 283.401,Z 463.346,A -85,B 0,C 180,E1 -16999.28,E2 -16999.28} C_VEL
LIN {X 0,Y 282.782,Z 466.674,A -85,B 0,C 180,E1 -17001.422,E2 -17001.422} C_VEL
LIN {X 0,Y 282.388,Z 469.624,A -85,B 0,C 180,E1 -17004.285,E2 -17004.285} C_VEL
LIN {X 0,Y 282.369,Z 470.497,A -85,B 0,C 180,E1 -17005.716,E2 -17005.716} C_VEL
LIN {X 0,Y 282.428,Z 470.945,A -85,B 0,C 180,E1 -17007.145,E2 -17007.145} C_VEL
LIN {X 0,Y 282.501,Z 470.675,A -85,B 0,C 180,E1 -17009.998,E2 -17009.998} C_VEL
LIN {X 0,Y 282.465,Z 469.944,A -85,B 0,C 180,E1 -17011.423,E2 -17011.423} C_VEL
LIN {X 0,Y 282.466,Z 468.763,A -85,B 0,C 180,E1 -17012.85,E2 -17012.85} C_VEL
LIN {X 0,Y 282.475,Z 467.163,A -85,B 0,C 180,E1 -17014.278,E2 -17014.278} C_VEL
LIN {X 0,Y 282.51,Z 463.921,A -85,B 0,C 180,E1 -17016.424,E2 -17016.424} C_VEL
LIN {X 0,Y 282.747,Z 459.586,A -85,B 0,C 180,E1 -17018.574,E2 -17018.574} C_VEL
LIN {X 0,Y 283.189,Z 454.032,A -85,B 0,C 180,E1 -17020.724,E2 -17020.724} C_VEL
LIN {X 0,Y 283.996,Z 447.085,A -85,B 0,C 180,E1 -17022.865,E2 -17022.865} C_VEL
LIN {X 0,Y 284.859,Z 439.971,A -85,B 0,C 180,E1 -17024.644,E2 -17024.644} C_VEL
LIN {X 0,Y 285.863,Z 431.801,A -85,B 0,C 180,E1 -17026.336,E2 -17026.336} C_VEL
LIN {X 0,Y 287.216,Z 421.937,A -85,B 0,C 180,E1 -17027.99,E2 -17027.99} C_VEL
LIN {X 0,Y 288.465,Z 411.645,A -85,B 0,C 180,E1 -17029.383,E2 -17029.383} C_VEL
LIN {X 0,Y 289.774,Z 400.413,A -85,B 0,C 180,E1 -17030.585,E2 -17030.585} C_VEL
LIN {X 0,Y 290.961,Z 389.076,A -85,B 0,C 180,E1 -17031.517,E2 -17031.517} C_VEL
LIN {X 0,Y 291.946,Z 376.319,A -85,B 0,C 180,E1 -17032.276,E2 -17032.276} C_VEL
LIN {X 0,Y 292.621,Z 362.77,A -85,B 0,C 180,E1 -17032.784,E2 -17032.784} C_VEL
LIN {X 0,Y 293.833,Z 303.65,A -85,B 0,C 180,E1 -17034.232,E2 -17034.232} C_VEL
LIN {X 0,Y 288.02,Z 258.035,A -85,B 0,C 180,E1 -17035.846,E2 -17035.846} C_VEL
LIN {X 0,Y 288.397,Z 254.566,A -85,B 0,C 180,E1 -17036.792,E2 -17036.792} C_VEL
LIN {X 0,Y 287.264,Z 247.97,A -85,B 0,C 180,E1 -17038.735,E2 -17038.735} C_VEL
LIN {X 0,Y 285.001,Z 237.28,A -85,B 0,C 180,E1 -17042.011,E2 -17042.011} C_VEL
LIN {X 0,Y 284.333,Z 234.067,A -85,B 0,C 180,E1 -17043.041,E2 -17043.041} C_VEL
LIN {X 0,Y 284.319,Z 234.072,A -85,B 0,C 180,E1 -17046.381,E2 -17046.381} C_VEL
LIN {X 0,Y 284.289,Z 234.076,A -85,B 0,C 180,E1 -17049.99,E2 -17049.99} C_VEL
LIN {X 0,Y 284.246,Z 234.078,A -85,B 0,C 180,E1 -17054.19,E2 -17054.19} C_VEL
LIN {X 0,Y 284.306,Z 234.071,A -85,B 0,C 180,E1 -17058.13,E2 -17058.13} C_VEL
LIN {X 0,Y 284.305,Z 234.072,A -85,B 0,C 180,E1 -17061.829,E2 -17061.829} C_VEL
LIN {X 0,Y 284.283,Z 234.073,A -85,B 0,C 180,E1 -17065.347,E2 -17065.347} C_VEL
LIN {X 0,Y 284.265,Z 234.073,A -85,B 0,C 180,E1 -17068.721,E2 -17068.721} C_VEL
LIN {X 0,Y 284.366,Z 234.06,A -85,B 0,C 180,E1 -17072.823,E2 -17072.823} C_VEL
LIN {X 0,Y 284.345,Z 234.062,A -85,B 0,C 180,E1 -17076.705,E2 -17076.705} C_VEL
LIN {X 0,Y 284.397,Z 234.057,A -85,B 0,C 180,E1 -17079.871,E2 -17079.871} C_VEL
LIN {X 0,Y 284.42,Z 234.054,A -85,B 0,C 180,E1 -17084.484,E2 -17084.484} C_VEL
LIN {X 0,Y 284.45,Z 234.047,A -85,B 0,C 180,E1 -17088.599,E2 -17088.599} C_VEL
LIN {X 0,Y 284.621,Z 234.031,A -85,B 0,C 180,E1 -17091.48,E2 -17091.48} C_VEL
LIN {X 0,Y 284.562,Z 234.035,A -85,B 0,C 180,E1 -17094.33,E2 -17094.33} C_VEL
LIN {X 0,Y 284.813,Z 233.994,A -85,B 0,C 180,E1 -17098.586,E2 -17098.586} C_VEL
LIN {X 0,Y 284.812,Z 233.998,A -85,B 0,C 180,E1 -17101.414,E2 -17101.414} C_VEL
LIN {X 0,Y 284.639,Z 234.03,A -85,B 0,C 180,E1 -17107.091,E2 -17107.091} C_VEL
LIN {X 0,Y 284.478,Z 234.044,A -85,B 0,C 180,E1 -17109.958,E2 -17109.958} C_VEL
LIN {X 0,Y 284.424,Z 234.054,A -85,B 0,C 180,E1 -17114.305,E2 -17114.305} C_VEL
LIN {X 0,Y 284.295,Z 234.07,A -85,B 0,C 180,E1 -17118.745,E2 -17118.745} C_VEL
LIN {X 0,Y 284.295,Z 234.07,A -85,B 0,C 180,E1 -17123.299,E2 -17123.299} C_VEL
LIN {X 0,Y 284.345,Z 234.058,A -85,B 0,C 180,E1 -17127.169,E2 -17127.169} C_VEL
LIN {X 0,Y 284.253,Z 234.062,A -85,B 0,C 180,E1 -17131.279,E2 -17131.279} C_VEL
LIN {X 0,Y 284.311,Z 234.066,A -85,B 0,C 180,E1 -17135.351,E2 -17135.351} C_VEL
LIN {X 0,Y 284.283,Z 234.073,A -85,B 0,C 180,E1 -17138.173,E2 -17138.173} C_VEL
LIN {X 0,Y 284.243,Z 234.071,A -85,B 0,C 180,E1 -17142.128,E2 -17142.128} C_VEL
LIN {X 0,Y 284.232,Z 234.078,A -85,B 0,C 180,E1 -17146.193,E2 -17146.193} C_VEL
LIN {X 0,Y 284.286,Z 234.074,A -85,B 0,C 180,E1 -17150.028,E2 -17150.028} C_VEL
LIN {X 0,Y 284.311,Z 234.064,A -85,B 0,C 180,E1 -17153.618,E2 -17153.618} C_VEL
LIN {X 0,Y 284.291,Z 234.07,A -85,B 0,C 180,E1 -17157.194,E2 -17157.194} C_VEL
LIN {X 0,Y 284.341,Z 234.065,A -85,B 0,C 180,E1 -17160.38,E2 -17160.38} C_VEL
LIN {X 0,Y 284.363,Z 234.063,A -85,B 0,C 180,E1 -17163.591,E2 -17163.591} C_VEL
LIN {X 0,Y 284.322,Z 234.067,A -85,B 0,C 180,E1 -17166.708,E2 -17166.708} C_VEL
LIN {X 0,Y 284.367,Z 234.066,A -85,B 0,C 180,E1 -17169.908,E2 -17169.908} C_VEL
LIN {X 0,Y 284.441,Z 234.056,A -85,B 0,C 180,E1 -17174.496,E2 -17174.496} C_VEL
LIN {X 0,Y 284.507,Z 234.047,A -85,B 0,C 180,E1 -17178.966,E2 -17178.966} C_VEL
LIN {X 0,Y 291.991,Z 254.548,A -85,B 0,C 180,E1 -17180.095,E2 -17180.095} C_VEL
LIN {X 0,Y 294.667,Z 263.566,A -85,B 0,C 180,E1 -17180.524,E2 -17180.524} C_VEL
LIN {X 0,Y 292.815,Z 340.891,A -85,B 0,C 180,E1 -17182.417,E2 -17182.417} C_VEL
LIN {X 0,Y 292.204,Z 354.19,A -85,B 0,C 180,E1 -17183.009,E2 -17183.009} C_VEL
LIN {X 0,Y 291.287,Z 366.962,A -85,B 0,C 180,E1 -17183.857,E2 -17183.857} C_VEL
LIN {X 0,Y 290.237,Z 379.096,A -85,B 0,C 180,E1 -17184.967,E2 -17184.967} C_VEL
LIN {X 0,Y 289.01,Z 390.826,A -85,B 0,C 180,E1 -17186.371,E2 -17186.371} C_VEL
LIN {X 0,Y 287.721,Z 401.022,A -85,B 0,C 180,E1 -17187.903,E2 -17187.903} C_VEL
LIN {X 0,Y 286.427,Z 410.379,A -85,B 0,C 180,E1 -17189.651,E2 -17189.651} C_VEL
LIN {X 0,Y 285.18,Z 419.424,A -85,B 0,C 180,E1 -17191.768,E2 -17191.768} C_VEL
LIN {X 0,Y 284.213,Z 426.713,A -85,B 0,C 180,E1 -17193.901,E2 -17193.901} C_VEL
LIN {X 0,Y 283.602,Z 431.634,A -85,B 0,C 180,E1 -17195.691,E2 -17195.691} C_VEL
LIN {X 0,Y 283.051,Z 436.421,A -85,B 0,C 180,E1 -17197.851,E2 -17197.851} C_VEL
LIN {X 0,Y 282.636,Z 440.09,A -85,B 0,C 180,E1 -17200.026,E2 -17200.026} C_VEL
LIN {X 0,Y 282.45,Z 441.976,A -85,B 0,C 180,E1 -17201.483,E2 -17201.483} C_VEL
LIN {X 0,Y 282.332,Z 444.082,A -85,B 0,C 180,E1 -17203.878,E2 -17203.878} C_VEL
LIN {X 0,Y 282.279,Z 445.002,A -85,B 0,C 180,E1 -17205.896,E2 -17205.896} C_VEL
LIN {X 0,Y 282.416,Z 445.154,A -85,B 0,C 180,E1 -17207.376,E2 -17207.376} C_VEL
LIN {X 0,Y 282.678,Z 444.802,A -85,B 0,C 180,E1 -17209.134,E2 -17209.134} C_VEL
LIN {X 0,Y 283.265,Z 443.101,A -85,B 0,C 180,E1 -17211.849,E2 -17211.849} C_VEL
LIN {X 0,Y 283.936,Z 441.098,A -85,B 0,C 180,E1 -17213.678,E2 -17213.678} C_VEL
LIN {X 0,Y 285.141,Z 436.919,A -85,B 0,C 180,E1 -17216.337,E2 -17216.337} C_VEL
LIN {X 0,Y 286.557,Z 432.048,A -85,B 0,C 180,E1 -17218.571,E2 -17218.571} C_VEL
LIN {X 0,Y 288.27,Z 425.788,A -85,B 0,C 180,E1 -17220.795,E2 -17220.795} C_VEL
LIN {X 0,Y 290.369,Z 417.9,A -85,B 0,C 180,E1 -17222.996,E2 -17222.996} C_VEL
LIN {X 0,Y 292.389,Z 409.687,A -85,B 0,C 180,E1 -17224.81,E2 -17224.81} C_VEL
LIN {X 0,Y 294.626,Z 399.529,A -85,B 0,C 180,E1 -17226.608,E2 -17226.608} C_VEL
LIN {X 0,Y 296.717,Z 389.503,A -85,B 0,C 180,E1 -17228.011,E2 -17228.011} C_VEL
LIN {X 0,Y 298.512,Z 378.6,A -85,B 0,C 180,E1 -17229.239,E2 -17229.239} C_VEL
LIN {X 0,Y 300.131,Z 366.2,A -85,B 0,C 180,E1 -17230.305,E2 -17230.305} C_VEL
LIN {X 0,Y 301.389,Z 353.558,A -85,B 0,C 180,E1 -17231.095,E2 -17231.095} C_VEL
LIN {X 0,Y 302.229,Z 340.528,A -85,B 0,C 180,E1 -17231.628,E2 -17231.628} C_VEL
LIN {X 0,Y 304.625,Z 274.499,A -85,B 0,C 180,E1 -17233.206,E2 -17233.206} C_VEL
LIN {X 0,Y 298.599,Z 261.014,A -85,B 0,C 180,E1 -17234.364,E2 -17234.364} C_VEL
LIN {X 0,Y 289.379,Z 243.471,A -85,B 0,C 180,E1 -17236.178,E2 -17236.178} C_VEL
LIN {X 0,Y 284.688,Z 235.409,A -85,B 0,C 180,E1 -17237.162,E2 -17237.162} C_VEL
LIN {X 0,Y 284.357,Z 234.062,A -85,B 0,C 180,E1 -17237.781,E2 -17237.781} C_VEL
LIN {X 0,Y 284.322,Z 234.065,A -85,B 0,C 180,E1 -17241.964,E2 -17241.964} C_VEL
LIN {X 0,Y 284.3,Z 234.064,A -85,B 0,C 180,E1 -17245.35,E2 -17245.35} C_VEL
LIN {X 0,Y 284.264,Z 234.067,A -85,B 0,C 180,E1 -17248.096,E2 -17248.096} C_VEL
LIN {X 0,Y 283.607,Z 234.154,A -85,B 0,C 180,E1 -17249.279,E2 -17249.279} C_VEL
LIN {X 0,Y 280.767,Z 234.501,A -85,B 0,C 180,E1 -17251.207,E2 -17251.207} C_VEL
LIN {X 0,Y 278.371,Z 234.806,A -85,B 0,C 180,E1 -17252.773,E2 -17252.773} C_VEL
LIN {X 0,Y 277.367,Z 234.928,A -85,B 0,C 180,E1 -17253.986,E2 -17253.986} C_VEL
LIN {X 0,Y 277.298,Z 234.933,A -85,B 0,C 180,E1 -17254.397,E2 -17254.397} C_VEL
LIN {X 0,Y 277.273,Z 234.941,A -85,B 0,C 180,E1 -17257.654,E2 -17257.654} C_VEL
LIN {X 0,Y 277.333,Z 234.937,A -85,B 0,C 180,E1 -17260.766,E2 -17260.766} C_VEL
LIN {X 0,Y 277.413,Z 234.931,A -85,B 0,C 180,E1 -17265.325,E2 -17265.325} C_VEL
LIN {X 0,Y 277.445,Z 234.925,A -85,B 0,C 180,E1 -17269.787,E2 -17269.787} C_VEL
LIN {X 0,Y 277.62,Z 234.893,A -85,B 0,C 180,E1 -17272.729,E2 -17272.729} C_VEL
LIN {X 0,Y 277.801,Z 234.875,A -85,B 0,C 180,E1 -17278.551,E2 -17278.551} C_VEL
LIN {X 0,Y 277.801,Z 234.865,A -85,B 0,C 180,E1 -17281.45,E2 -17281.45} C_VEL
LIN {X 0,Y 277.588,Z 234.898,A -85,B 0,C 180,E1 -17287.273,E2 -17287.273} C_VEL
LIN {X 0,Y 277.44,Z 234.909,A -85,B 0,C 180,E1 -17290.214,E2 -17290.214} C_VEL
LIN {X 0,Y 277.395,Z 234.918,A -85,B 0,C 180,E1 -17294.677,E2 -17294.677} C_VEL
LIN {X 0,Y 277.269,Z 234.936,A -85,B 0,C 180,E1 -17299.24,E2 -17299.24} C_VEL
LIN {X 0,Y 277.27,Z 234.939,A -85,B 0,C 180,E1 -17303.926,E2 -17303.926} C_VEL
LIN {X 0,Y 277.259,Z 234.94,A -85,B 0,C 180,E1 -17307.483,E2 -17307.483} C_VEL
LIN {X 0,Y 277.24,Z 234.945,A -85,B 0,C 180,E1 -17310.474,E2 -17310.474} C_VEL
LIN {X 0,Y 277.231,Z 234.948,A -85,B 0,C 180,E1 -17313.899,E2 -17313.899} C_VEL
LIN {X 0,Y 277.248,Z 234.944,A -85,B 0,C 180,E1 -17317.473,E2 -17317.473} C_VEL
LIN {X 0,Y 277.195,Z 234.936,A -85,B 0,C 180,E1 -17321.24,E2 -17321.24} C_VEL
LIN {X 0,Y 277.191,Z 234.955,A -85,B 0,C 180,E1 -17325.229,E2 -17325.229} C_VEL
LIN {X 0,Y 277.231,Z 235.063,A -85,B 0,C 180,E1 -17329.433,E2 -17329.433} C_VEL
LIN {X 0,Y 280.017,Z 244.824,A -85,B 0,C 180,E1 -17333.433,E2 -17333.433} C_VEL
LIN {X 0,Y 281.955,Z 252.484,A -85,B 0,C 180,E1 -17336.323,E2 -17336.323} C_VEL
LIN {X 0,Y 282.849,Z 256.36,A -85,B 0,C 180,E1 -17337.652,E2 -17337.652} C_VEL
LIN {X 0,Y 290.135,Z 271.788,A -85,B 0,C 180,E1 -17339.211,E2 -17339.211} C_VEL
LIN {X 0,Y 291.882,Z 276.144,A -85,B 0,C 180,E1 -17339.587,E2 -17339.587} C_VEL
LIN {X 0,Y 296.269,Z 299.537,A -85,B 0,C 180,E1 -17340.865,E2 -17340.865} C_VEL
LIN {X 0,Y 297.543,Z 310.385,A -85,B 0,C 180,E1 -17341.341,E2 -17341.341} C_VEL
LIN {X 0,Y 295.461,Z 366.179,A -85,B 0,C 180,E1 -17342.724,E2 -17342.724} C_VEL
LIN {X 0,Y 294.243,Z 379.521,A -85,B 0,C 180,E1 -17343.299,E2 -17343.299} C_VEL
LIN {X 0,Y 292.636,Z 391.979,A -85,B 0,C 180,E1 -17344.1,E2 -17344.1} C_VEL
LIN {X 0,Y 290.589,Z 403.914,A -85,B 0,C 180,E1 -17345.151,E2 -17345.151} C_VEL
LIN {X 0,Y 288.245,Z 415.346,A -85,B 0,C 180,E1 -17346.468,E2 -17346.468} C_VEL
LIN {X 0,Y 285.934,Z 425.669,A -85,B 0,C 180,E1 -17347.986,E2 -17347.986} C_VEL
LIN {X 0,Y 283.628,Z 434.989,A -85,B 0,C 180,E1 -17349.701,E2 -17349.701} C_VEL
LIN {X 0,Y 281.723,Z 442.615,A -85,B 0,C 180,E1 -17351.437,E2 -17351.437} C_VEL
LIN {X 0,Y 279.786,Z 450.223,A -85,B 0,C 180,E1 -17353.584,E2 -17353.584} C_VEL
LIN {X 0,Y 277.834,Z 457.241,A -85,B 0,C 180,E1 -17356.094,E2 -17356.094} C_VEL
LIN {X 0,Y 276.666,Z 461.921,A -85,B 0,C 180,E1 -17358.273,E2 -17358.273} C_VEL
LIN {X 0,Y 275.921,Z 465.52,A -85,B 0,C 180,E1 -17360.468,E2 -17360.468} C_VEL
LIN {X 0,Y 275.454,Z 468.135,A -85,B 0,C 180,E1 -17362.669,E2 -17362.669} C_VEL
LIN {X 0,Y 275.332,Z 469.652,A -85,B 0,C 180,E1 -17364.564,E2 -17364.564} C_VEL
LIN {X 0,Y 275.353,Z 470.63,A -85,B 0,C 180,E1 -17367.072,E2 -17367.072} C_VEL
LIN {X 0,Y 275.351,Z 470.662,A -85,B 0,C 180,E1 -17368.535,E2 -17368.535} C_VEL
LIN {X 0,Y 275.416,Z 470.308,A -85,B 0,C 180,E1 -17369.997,E2 -17369.997} C_VEL
LIN {X 0,Y 275.384,Z 469.53,A -85,B 0,C 180,E1 -17371.46,E2 -17371.46} C_VEL
LIN {X 0,Y 275.394,Z 468.316,A -85,B 0,C 180,E1 -17372.923,E2 -17372.923} C_VEL
LIN {X 0,Y 275.385,Z 465.078,A -85,B 0,C 180,E1 -17375.55,E2 -17375.55} C_VEL
LIN {X 0,Y 275.58,Z 460.609,A -85,B 0,C 180,E1 -17378.06,E2 -17378.06} C_VEL
LIN {X 0,Y 276.056,Z 454.391,A -85,B 0,C 180,E1 -17380.633,E2 -17380.633} C_VEL
LIN {X 0,Y 276.841,Z 447.594,A -85,B 0,C 180,E1 -17382.83,E2 -17382.83} C_VEL
LIN {X 0,Y 277.962,Z 439.142,A -85,B 0,C 180,E1 -17385.016,E2 -17385.016} C_VEL
LIN {X 0,Y 279.186,Z 429.768,A -85,B 0,C 180,E1 -17386.944,E2 -17386.944} C_VEL
LIN {X 0,Y 280.568,Z 419.636,A -85,B 0,C 180,E1 -17388.621,E2 -17388.621} C_VEL
LIN {X 0,Y 281.94,Z 408.931,A -85,B 0,C 180,E1 -17390.04,E2 -17390.04} C_VEL
LIN {X 0,Y 283.353,Z 396.979,A -85,B 0,C 180,E1 -17391.264,E2 -17391.264} C_VEL
LIN {X 0,Y 284.563,Z 384.533,A -85,B 0,C 180,E1 -17392.216,E2 -17392.216} C_VEL
LIN {X 0,Y 285.501,Z 371.736,A -85,B 0,C 180,E1 -17392.903,E2 -17392.903} C_VEL
LIN {X 0,Y 286.012,Z 357.687,A -85,B 0,C 180,E1 -17393.351,E2 -17393.351} C_VEL
LIN {X 0,Y 287.153,Z 304.548,A -85,B 0,C 180,E1 -17394.673,E2 -17394.673} C_VEL
LIN {X 0,Y 281.434,Z 259.259,A -85,B 0,C 180,E1 -17396.312,E2 -17396.312} C_VEL
LIN {X 0,Y 281.241,Z 257.549,A -85,B 0,C 180,E1 -17396.424,E2 -17396.424} C_VEL
LIN {X 0,Y 281.191,Z 253.7,A -85,B 0,C 180,E1 -17397.535,E2 -17397.535} C_VEL
LIN {X 0,Y 278.633,Z 241.199,A -85,B 0,C 180,E1 -17401.409,E2 -17401.409} C_VEL
LIN {X 0,Y 277.275,Z 234.948,A -85,B 0,C 180,E1 -17403.494,E2 -17403.494} C_VEL
LIN {X 0,Y 277.256,Z 234.951,A -85,B 0,C 180,E1 -17407.464,E2 -17407.464} C_VEL
LIN {X 0,Y 277.192,Z 234.956,A -85,B 0,C 180,E1 -17411.232,E2 -17411.232} C_VEL
LIN {X 0,Y 277.21,Z 234.952,A -85,B 0,C 180,E1 -17415.216,E2 -17415.216} C_VEL
LIN {X 0,Y 277.27,Z 234.948,A -85,B 0,C 180,E1 -17419.491,E2 -17419.491} C_VEL
LIN {X 0,Y 277.258,Z 234.946,A -85,B 0,C 180,E1 -17422.529,E2 -17422.529} C_VEL
LIN {X 0,Y 277.22,Z 234.951,A -85,B 0,C 180,E1 -17426.1,E2 -17426.1} C_VEL
LIN {X 0,Y 277.234,Z 234.953,A -85,B 0,C 180,E1 -17429.535,E2 -17429.535} C_VEL
LIN {X 0,Y 277.327,Z 234.937,A -85,B 0,C 180,E1 -17432.86,E2 -17432.86} C_VEL
LIN {X 0,Y 277.311,Z 234.939,A -85,B 0,C 180,E1 -17436.077,E2 -17436.077} C_VEL
LIN {X 0,Y 277.336,Z 234.936,A -85,B 0,C 180,E1 -17440.765,E2 -17440.765} C_VEL
LIN {X 0,Y 277.379,Z 234.936,A -85,B 0,C 180,E1 -17445.322,E2 -17445.322} C_VEL
LIN {X 0,Y 277.469,Z 234.92,A -85,B 0,C 180,E1 -17449.787,E2 -17449.787} C_VEL
LIN {X 0,Y 277.615,Z 234.903,A -85,B 0,C 180,E1 -17452.728,E2 -17452.728} C_VEL
LIN {X 0,Y 277.78,Z 234.869,A -85,B 0,C 180,E1 -17458.55,E2 -17458.55} C_VEL
LIN {X 0,Y 277.779,Z 234.873,A -85,B 0,C 180,E1 -17461.449,E2 -17461.449} C_VEL
LIN {X 0,Y 277.594,Z 234.906,A -85,B 0,C 180,E1 -17467.272,E2 -17467.272} C_VEL
LIN {X 0,Y 277.421,Z 234.924,A -85,B 0,C 180,E1 -17470.214,E2 -17470.214} C_VEL
LIN {X 0,Y 277.371,Z 234.935,A -85,B 0,C 180,E1 -17474.677,E2 -17474.677} C_VEL
LIN {X 0,Y 277.248,Z 234.944,A -85,B 0,C 180,E1 -17479.24,E2 -17479.24} C_VEL
LIN {X 0,Y 277.259,Z 234.946,A -85,B 0,C 180,E1 -17483.926,E2 -17483.926} C_VEL
LIN {X 0,Y 277.275,Z 234.937,A -85,B 0,C 180,E1 -17487.5,E2 -17487.5} C_VEL
LIN {X 0,Y 277.217,Z 234.937,A -85,B 0,C 180,E1 -17490.476,E2 -17490.476} C_VEL
LIN {X 0,Y 277.216,Z 234.946,A -85,B 0,C 180,E1 -17493.899,E2 -17493.899} C_VEL
LIN {X 0,Y 277.238,Z 234.948,A -85,B 0,C 180,E1 -17497.473,E2 -17497.473} C_VEL
LIN {X 0,Y 277.183,Z 234.948,A -85,B 0,C 180,E1 -17501.241,E2 -17501.241} C_VEL
LIN {X 0,Y 277.177,Z 234.952,A -85,B 0,C 180,E1 -17505.231,E2 -17505.231} C_VEL
LIN {X 0,Y 277.201,Z 234.953,A -85,B 0,C 180,E1 -17509.517,E2 -17509.517} C_VEL
LIN {X 0,Y 277.245,Z 234.943,A -85,B 0,C 180,E1 -17512.534,E2 -17512.534} C_VEL
LIN {X 0,Y 277.23,Z 234.954,A -85,B 0,C 180,E1 -17516.108,E2 -17516.108} C_VEL
LIN {X 0,Y 277.247,Z 234.944,A -85,B 0,C 180,E1 -17519.543,E2 -17519.543} C_VEL
LIN {X 0,Y 277.344,Z 234.936,A -85,B 0,C 180,E1 -17522.868,E2 -17522.868} C_VEL
LIN {X 0,Y 277.286,Z 234.946,A -85,B 0,C 180,E1 -17526.081,E2 -17526.081} C_VEL
LIN {X 0,Y 277.303,Z 234.942,A -85,B 0,C 180,E1 -17530.768,E2 -17530.768} C_VEL
LIN {X 0,Y 277.403,Z 234.934,A -85,B 0,C 180,E1 -17535.328,E2 -17535.328} C_VEL
LIN {X 0,Y 277.454,Z 234.927,A -85,B 0,C 180,E1 -17538.424,E2 -17538.424} C_VEL
LIN {X 0,Y 279.163,Z 239.516,A -85,B 0,C 180,E1 -17538.699,E2 -17538.699} C_VEL
LIN {X 0,Y 284.702,Z 254.186,A -85,B 0,C 180,E1 -17539.539,E2 -17539.539} C_VEL
LIN {X 0,Y 288.099,Z 264.99,A -85,B 0,C 180,E1 -17540.083,E2 -17540.083} C_VEL
LIN {X 0,Y 286.001,Z 342.171,A -85,B 0,C 180,E1 -17542.014,E2 -17542.014} C_VEL
LIN {X 0,Y 285.388,Z 355.858,A -85,B 0,C 180,E1 -17542.664,E2 -17542.664} C_VEL
LIN {X 0,Y 284.503,Z 367.178,A -85,B 0,C 180,E1 -17543.443,E2 -17543.443} C_VEL
LIN {X 0,Y 283.504,Z 378.543,A -85,B 0,C 180,E1 -17544.491,E2 -17544.491} C_VEL
LIN {X 0,Y 282.211,Z 390.562,A -85,B 0,C 180,E1 -17545.943,E2 -17545.943} C_VEL
LIN {X 0,Y 280.88,Z 400.762,A -85,B 0,C 180,E1 -17547.493,E2 -17547.493} C_VEL
LIN {X 0,Y 279.552,Z 410.25,A -85,B 0,C 180,E1 -17549.282,E2 -17549.282} C_VEL
LIN {X 0,Y 278.234,Z 419.376,A -85,B 0,C 180,E1 -17551.45,E2 -17551.45} C_VEL
LIN {X 0,Y 277.223,Z 426.73,A -85,B 0,C 180,E1 -17553.636,E2 -17553.636} C_VEL
LIN {X 0,Y 276.487,Z 432.622,A -85,B 0,C 180,E1 -17555.838,E2 -17555.838} C_VEL
LIN {X 0,Y 275.918,Z 437.268,A -85,B 0,C 180,E1 -17558.055,E2 -17558.055} C_VEL
LIN {X 0,Y 275.519,Z 440.809,A -85,B 0,C 180,E1 -17560.287,E2 -17560.287} C_VEL
LIN {X 0,Y 275.323,Z 442.579,A -85,B 0,C 180,E1 -17561.785,E2 -17561.785} C_VEL
LIN {X 0,Y 275.227,Z 444.424,A -85,B 0,C 180,E1 -17563.991,E2 -17563.991} C_VEL
LIN {X 0,Y 275.222,Z 445.384,A -85,B 0,C 180,E1 -17566.315,E2 -17566.315} C_VEL
LIN {X 0,Y 275.384,Z 445.46,A -85,B 0,C 180,E1 -17567.834,E2 -17567.834} C_VEL
LIN {X 0,Y 275.619,Z 445.134,A -85,B 0,C 180,E1 -17569.36,E2 -17569.36} C_VEL
LIN {X 0,Y 275.922,Z 444.389,A -85,B 0,C 180,E1 -17570.892,E2 -17570.892} C_VEL
LIN {X 0,Y 276.367,Z 443.164,A -85,B 0,C 180,E1 -17572.424,E2 -17572.424} C_VEL
LIN {X 0,Y 277.263,Z 440.501,A -85,B 0,C 180,E1 -17574.723,E2 -17574.723} C_VEL
LIN {X 0,Y 278.44,Z 436.721,A -85,B 0,C 180,E1 -17577.022,E2 -17577.022} C_VEL
LIN {X 0,Y 280.002,Z 431.707,A -85,B 0,C 180,E1 -17579.304,E2 -17579.304} C_VEL
LIN {X 0,Y 281.859,Z 425.291,A -85,B 0,C 180,E1 -17581.575,E2 -17581.575} C_VEL
LIN {X 0,Y 284.109,Z 417.135,A -85,B 0,C 180,E1 -17583.819,E2 -17583.819} C_VEL
LIN {X 0,Y 286.447,Z 407.933,A -85,B 0,C 180,E1 -17585.815,E2 -17585.815} C_VEL
LIN {X 0,Y 288.65,Z 398.256,A -85,B 0,C 180,E1 -17587.494,E2 -17587.494} C_VEL
LIN {X 0,Y 290.847,Z 387.786,A -85,B 0,C 180,E1 -17588.921,E2 -17588.921} C_VEL
LIN {X 0,Y 292.593,Z 377.137,A -85,B 0,C 180,E1 -17590.089,E2 -17590.089} C_VEL
LIN {X 0,Y 294.178,Z 365.538,A -85,B 0,C 180,E1 -17591.069,E2 -17591.069} C_VEL
LIN {X 0,Y 295.414,Z 353.028,A -85,B 0,C 180,E1 -17591.848,E2 -17591.848} C_VEL
LIN {X 0,Y 296.225,Z 340.543,A -85,B 0,C 180,E1 -17592.351,E2 -17592.351} C_VEL
LIN {X 0,Y 298.657,Z 276.493,A -85,B 0,C 180,E1 -17593.906,E2 -17593.906} C_VEL
LIN {X 0,Y 292.469,Z 262.861,A -85,B 0,C 180,E1 -17595.146,E2 -17595.146} C_VEL
LIN {X 0,Y 284.486,Z 247.742,A -85,B 0,C 180,E1 -17596.783,E2 -17596.783} C_VEL
LIN {X 0,Y 279.023,Z 238.739,A -85,B 0,C 180,E1 -17597.941,E2 -17597.941} C_VEL
LIN {X 0,Y 277.597,Z 236.296,A -85,B 0,C 180,E1 -17598.257,E2 -17598.257} C_VEL
LIN {X 0,Y 277.382,Z 235.559,A -85,B 0,C 180,E1 -17598.44,E2 -17598.44} C_VEL
LIN {X 0,Y 277.286,Z 234.947,A -85,B 0,C 180,E1 -17598.778,E2 -17598.778} C_VEL
LIN {X 0,Y 277.276,Z 234.941,A -85,B 0,C 180,E1 -17602.533,E2 -17602.533} C_VEL
LIN {X 0,Y 277.238,Z 234.947,A -85,B 0,C 180,E1 -17606.104,E2 -17606.104} C_VEL
LIN {X 0,Y 277.252,Z 234.946,A -85,B 0,C 180,E1 -17609.538,E2 -17609.538} C_VEL
LIN {X 0,Y 277.347,Z 234.933,A -85,B 0,C 180,E1 -17612.863,E2 -17612.863} C_VEL
LIN {X 0,Y 277.298,Z 234.933,A -85,B 0,C 180,E1 -17614.397,E2 -17614.397} C_VEL
LIN {X 0,Y 276.668,Z 235.015,A -85,B 0,C 180,E1 -17615.609,E2 -17615.609} C_VEL
LIN {X 0,Y 273.836,Z 235.372,A -85,B 0,C 180,E1 -17617.584,E2 -17617.584} C_VEL
LIN {X 0,Y 271.405,Z 235.674,A -85,B 0,C 180,E1 -17619.189,E2 -17619.189} C_VEL
LIN {X 0,Y 270.351,Z 235.807,A -85,B 0,C 180,E1 -17620.432,E2 -17620.432} C_VEL
LIN {X 0,Y 270.26,Z 235.812,A -85,B 0,C 180,E1 -17620.854,E2 -17620.854} C_VEL
LIN {X 0,Y 270.382,Z 235.804,A -85,B 0,C 180,E1 -17624.935,E2 -17624.935} C_VEL
LIN {X 0,Y 270.397,Z 235.804,A -85,B 0,C 180,E1 -17629.518,E2 -17629.518} C_VEL
LIN {X 0,Y 270.576,Z 235.769,A -85,B 0,C 180,E1 -17632.538,E2 -17632.538} C_VEL
LIN {X 0,Y 270.768,Z 235.751,A -85,B 0,C 180,E1 -17638.513,E2 -17638.513} C_VEL
LIN {X 0,Y 270.767,Z 235.741,A -85,B 0,C 180,E1 -17641.488,E2 -17641.488} C_VEL
LIN {X 0,Y 270.55,Z 235.777,A -85,B 0,C 180,E1 -17647.463,E2 -17647.463} C_VEL
LIN {X 0,Y 270.374,Z 235.789,A -85,B 0,C 180,E1 -17650.484,E2 -17650.484} C_VEL
LIN {X 0,Y 270.355,Z 235.795,A -85,B 0,C 180,E1 -17655.068,E2 -17655.068} C_VEL
LIN {X 0,Y 270.21,Z 235.817,A -85,B 0,C 180,E1 -17659.763,E2 -17659.763} C_VEL
LIN {X 0,Y 270.214,Z 235.822,A -85,B 0,C 180,E1 -17664.592,E2 -17664.592} C_VEL
LIN {X 0,Y 270.187,Z 235.822,A -85,B 0,C 180,E1 -17667.919,E2 -17667.919} C_VEL
LIN {X 0,Y 270.161,Z 235.825,A -85,B 0,C 180,E1 -17671.352,E2 -17671.352} C_VEL
LIN {X 0,Y 270.187,Z 235.824,A -85,B 0,C 180,E1 -17674.908,E2 -17674.908} C_VEL
LIN {X 0,Y 270.193,Z 235.828,A -85,B 0,C 180,E1 -17678.712,E2 -17678.712} C_VEL
LIN {X 0,Y 270.157,Z 235.822,A -85,B 0,C 180,E1 -17683.249,E2 -17683.249} C_VEL
LIN {X 0,Y 270.148,Z 235.832,A -85,B 0,C 180,E1 -17687.438,E2 -17687.438} C_VEL
LIN {X 0,Y 270.158,Z 235.953,A -85,B 0,C 180,E1 -17688.381,E2 -17688.381} C_VEL
LIN {X 0,Y 272.702,Z 244.538,A -85,B 0,C 180,E1 -17692.097,E2 -17692.097} C_VEL
LIN {X 0,Y 275.088,Z 253.956,A -85,B 0,C 180,E1 -17695.802,E2 -17695.802} C_VEL
LIN {X 0,Y 275.539,Z 255.864,A -85,B 0,C 180,E1 -17696.464,E2 -17696.464} C_VEL
LIN {X 0,Y 282.466,Z 269.97,A -85,B 0,C 180,E1 -17698.026,E2 -17698.026} C_VEL
LIN {X 0,Y 286.328,Z 278.717,A -85,B 0,C 180,E1 -17698.876,E2 -17698.876} C_VEL
LIN {X 0,Y 290.588,Z 302.052,A -85,B 0,C 180,E1 -17700.182,E2 -17700.182} C_VEL
LIN {X 0,Y 291.618,Z 311.28,A -85,B 0,C 180,E1 -17700.596,E2 -17700.596} C_VEL
LIN {X 0,Y 289.453,Z 365.716,A -85,B 0,C 180,E1 -17701.965,E2 -17701.965} C_VEL
LIN {X 0,Y 288.26,Z 379.028,A -85,B 0,C 180,E1 -17702.552,E2 -17702.552} C_VEL
LIN {X 0,Y 286.485,Z 392.067,A -85,B 0,C 180,E1 -17703.403,E2 -17703.403} C_VEL
LIN {X 0,Y 284.206,Z 404.671,A -85,B 0,C 180,E1 -17704.554,E2 -17704.554} C_VEL
LIN {X 0,Y 281.77,Z 415.907,A -85,B 0,C 180,E1 -17705.893,E2 -17705.893} C_VEL
LIN {X 0,Y 279.381,Z 426.06,A -85,B 0,C 180,E1 -17707.441,E2 -17707.441} C_VEL
LIN {X 0,Y 276.977,Z 435.221,A -85,B 0,C 180,E1 -17709.191,E2 -17709.191} C_VEL
LIN {X 0,Y 274.827,Z 443.329,A -85,B 0,C 180,E1 -17711.118,E2 -17711.118} C_VEL
LIN {X 0,Y 272.629,Z 451.399,A -85,B 0,C 180,E1 -17713.526,E2 -17713.526} C_VEL
LIN {X 0,Y 270.94,Z 457.22,A -85,B 0,C 180,E1 -17715.733,E2 -17715.733} C_VEL
LIN {X 0,Y 269.669,Z 461.833,A -85,B 0,C 180,E1 -17717.964,E2 -17717.964} C_VEL
LIN {X 0,Y 268.892,Z 465.373,A -85,B 0,C 180,E1 -17720.217,E2 -17720.217} C_VEL
LIN {X 0,Y 268.378,Z 467.928,A -85,B 0,C 180,E1 -17722.474,E2 -17722.474} C_VEL
LIN {X 0,Y 268.226,Z 469.53,A -85,B 0,C 180,E1 -17724.671,E2 -17724.671} C_VEL
LIN {X 0,Y 268.257,Z 470.314,A -85,B 0,C 180,E1 -17726.994,E2 -17726.994} C_VEL
LIN {X 0,Y 268.273,Z 470.321,A -85,B 0,C 180,E1 -17728.496,E2 -17728.496} C_VEL
LIN {X 0,Y 268.333,Z 469.939,A -85,B 0,C 180,E1 -17729.997,E2 -17729.997} C_VEL
LIN {X 0,Y 268.306,Z 469.11,A -85,B 0,C 180,E1 -17731.498,E2 -17731.498} C_VEL
LIN {X 0,Y 268.323,Z 467.87,A -85,B 0,C 180,E1 -17733,E2 -17733} C_VEL
LIN {X 0,Y 268.288,Z 464.898,A -85,B 0,C 180,E1 -17735.47,E2 -17735.47} C_VEL
LIN {X 0,Y 268.436,Z 461.491,A -85,B 0,C 180,E1 -17737.519,E2 -17737.519} C_VEL
LIN {X 0,Y 268.771,Z 456.631,A -85,B 0,C 180,E1 -17739.782,E2 -17739.782} C_VEL
LIN {X 0,Y 269.361,Z 450.474,A -85,B 0,C 180,E1 -17742.044,E2 -17742.044} C_VEL
LIN {X 0,Y 270.454,Z 442.819,A -85,B 0,C 180,E1 -17744.288,E2 -17744.288} C_VEL
LIN {X 0,Y 271.59,Z 434.971,A -85,B 0,C 180,E1 -17746.147,E2 -17746.147} C_VEL
LIN {X 0,Y 272.679,Z 426.564,A -85,B 0,C 180,E1 -17747.792,E2 -17747.792} C_VEL
LIN {X 0,Y 274.105,Z 415.967,A -85,B 0,C 180,E1 -17749.466,E2 -17749.466} C_VEL
LIN {X 0,Y 275.626,Z 404.37,A -85,B 0,C 180,E1 -17750.91,E2 -17750.91} C_VEL
LIN {X 0,Y 277.02,Z 392.189,A -85,B 0,C 180,E1 -17752.069,E2 -17752.069} C_VEL
LIN {X 0,Y 278.217,Z 378.607,A -85,B 0,C 180,E1 -17752.996,E2 -17752.996} C_VEL
LIN {X 0,Y 279.012,Z 366.032,A -85,B 0,C 180,E1 -17753.565,E2 -17753.565} C_VEL
LIN {X 0,Y 280.459,Z 305.075,A -85,B 0,C 180,E1 -17755.142,E2 -17755.142} C_VEL
LIN {X 0,Y 274.474,Z 257.948,A -85,B 0,C 180,E1 -17756.908,E2 -17756.908} C_VEL
LIN {X 0,Y 274.424,Z 257.341,A -85,B 0,C 180,E1 -17756.951,E2 -17756.951} C_VEL
LIN {X 0,Y 273.47,Z 251.29,A -85,B 0,C 180,E1 -17758.816,E2 -17758.816} C_VEL
LIN {X 0,Y 271.355,Z 241.069,A -85,B 0,C 180,E1 -17762.097,E2 -17762.097} C_VEL
LIN {X 0,Y 270.233,Z 235.827,A -85,B 0,C 180,E1 -17763.875,E2 -17763.875} C_VEL
LIN {X 0,Y 270.213,Z 235.828,A -85,B 0,C 180,E1 -17766.735,E2 -17766.735} C_VEL
LIN {X 0,Y 270.152,Z 235.833,A -85,B 0,C 180,E1 -17771.023,E2 -17771.023} C_VEL
LIN {X 0,Y 270.16,Z 235.831,A -85,B 0,C 180,E1 -17775.381,E2 -17775.381} C_VEL
LIN {X 0,Y 270.221,Z 235.826,A -85,B 0,C 180,E1 -17779.442,E2 -17779.442} C_VEL
LIN {X 0,Y 270.223,Z 235.825,A -85,B 0,C 180,E1 -17783.72,E2 -17783.72} C_VEL
LIN {X 0,Y 270.175,Z 235.827,A -85,B 0,C 180,E1 -17786.888,E2 -17786.888} C_VEL
LIN {X 0,Y 270.2,Z 235.824,A -85,B 0,C 180,E1 -17790.383,E2 -17790.383} C_VEL
LIN {X 0,Y 270.235,Z 235.823,A -85,B 0,C 180,E1 -17793.76,E2 -17793.76} C_VEL
LIN {X 0,Y 270.212,Z 235.824,A -85,B 0,C 180,E1 -17797.036,E2 -17797.036} C_VEL
LIN {X 0,Y 270.293,Z 235.813,A -85,B 0,C 180,E1 -17800.243,E2 -17800.243} C_VEL
LIN {X 0,Y 270.347,Z 235.809,A -85,B 0,C 180,E1 -17804.932,E2 -17804.932} C_VEL
LIN {X 0,Y 270.405,Z 235.801,A -85,B 0,C 180,E1 -17809.517,E2 -17809.517} C_VEL
LIN {X 0,Y 270.574,Z 235.779,A -85,B 0,C 180,E1 -17812.537,E2 -17812.537} C_VEL
LIN {X 0,Y 270.746,Z 235.743,A -85,B 0,C 180,E1 -17818.512,E2 -17818.512} C_VEL
LIN {X 0,Y 270.745,Z 235.747,A -85,B 0,C 180,E1 -17821.487,E2 -17821.487} C_VEL
LIN {X 0,Y 270.551,Z 235.782,A -85,B 0,C 180,E1 -17827.462,E2 -17827.462} C_VEL
LIN {X 0,Y 270.374,Z 235.803,A -85,B 0,C 180,E1 -17830.483,E2 -17830.483} C_VEL
LIN {X 0,Y 270.33,Z 235.812,A -85,B 0,C 180,E1 -17835.068,E2 -17835.068} C_VEL
LIN {X 0,Y 270.188,Z 235.822,A -85,B 0,C 180,E1 -17839.764,E2 -17839.764} C_VEL
LIN {X 0,Y 270.202,Z 235.828,A -85,B 0,C 180,E1 -17844.592,E2 -17844.592} C_VEL
LIN {X 0,Y 270.211,Z 235.817,A -85,B 0,C 180,E1 -17847.915,E2 -17847.915} C_VEL
LIN {X 0,Y 270.143,Z 235.817,A -85,B 0,C 180,E1 -17851.353,E2 -17851.353} C_VEL
LIN {X 0,Y 270.172,Z 235.828,A -85,B 0,C 180,E1 -17854.909,E2 -17854.909} C_VEL
LIN {X 0,Y 270.172,Z 235.829,A -85,B 0,C 180,E1 -17858.714,E2 -17858.714} C_VEL
LIN {X 0,Y 270.14,Z 235.82,A -85,B 0,C 180,E1 -17863.253,E2 -17863.253} C_VEL
LIN {X 0,Y 270.149,Z 235.832,A -85,B 0,C 180,E1 -17867.446,E2 -17867.446} C_VEL
LIN {X 0,Y 270.188,Z 235.822,A -85,B 0,C 180,E1 -17871.378,E2 -17871.378} C_VEL
LIN {X 0,Y 270.184,Z 235.827,A -85,B 0,C 180,E1 -17875.099,E2 -17875.099} C_VEL
LIN {X 0,Y 270.186,Z 235.823,A -85,B 0,C 180,E1 -17879.135,E2 -17879.135} C_VEL
LIN {X 0,Y 270.251,Z 235.823,A -85,B 0,C 180,E1 -17882.151,E2 -17882.151} C_VEL
LIN {X 0,Y 270.226,Z 235.825,A -85,B 0,C 180,E1 -17885.542,E2 -17885.542} C_VEL
LIN {X 0,Y 270.246,Z 235.823,A -85,B 0,C 180,E1 -17890.245,E2 -17890.245} C_VEL
LIN {X 0,Y 270.371,Z 235.809,A -85,B 0,C 180,E1 -17894.938,E2 -17894.938} C_VEL
LIN {X 0,Y 270.383,Z 235.81,A -85,B 0,C 180,E1 -17897.835,E2 -17897.835} C_VEL
LIN {X 0,Y 271.423,Z 238.719,A -85,B 0,C 180,E1 -17898.024,E2 -17898.024} C_VEL
LIN {X 0,Y 276.625,Z 251.533,A -85,B 0,C 180,E1 -17898.824,E2 -17898.824} C_VEL
LIN {X 0,Y 281.454,Z 266.47,A -85,B 0,C 180,E1 -17899.619,E2 -17899.619} C_VEL
LIN {X 0,Y 279.285,Z 342.133,A -85,B 0,C 180,E1 -17901.547,E2 -17901.547} C_VEL
LIN {X 0,Y 278.681,Z 355.19,A -85,B 0,C 180,E1 -17902.167,E2 -17902.167} C_VEL
LIN {X 0,Y 277.732,Z 367.319,A -85,B 0,C 180,E1 -17903.008,E2 -17903.008} C_VEL
LIN {X 0,Y 276.607,Z 379.542,A -85,B 0,C 180,E1 -17904.17,E2 -17904.17} C_VEL
LIN {X 0,Y 275.338,Z 391.093,A -85,B 0,C 180,E1 -17905.611,E2 -17905.611} C_VEL
LIN {X 0,Y 273.937,Z 401.532,A -85,B 0,C 180,E1 -17907.246,E2 -17907.246} C_VEL
LIN {X 0,Y 272.684,Z 410.072,A -85,B 0,C 180,E1 -17908.895,E2 -17908.895} C_VEL
LIN {X 0,Y 271.496,Z 417.94,A -85,B 0,C 180,E1 -17910.744,E2 -17910.744} C_VEL
LIN {X 0,Y 270.364,Z 425.613,A -85,B 0,C 180,E1 -17912.982,E2 -17912.982} C_VEL
LIN {X 0,Y 269.533,Z 431.778,A -85,B 0,C 180,E1 -17915.238,E2 -17915.238} C_VEL
LIN {X 0,Y 268.95,Z 436.67,A -85,B 0,C 180,E1 -17917.509,E2 -17917.509} C_VEL
LIN {X 0,Y 268.498,Z 440.441,A -85,B 0,C 180,E1 -17919.798,E2 -17919.798} C_VEL
LIN {X 0,Y 268.216,Z 443.176,A -85,B 0,C 180,E1 -17922.102,E2 -17922.102} C_VEL
LIN {X 0,Y 268.134,Z 444.769,A -85,B 0,C 180,E1 -17924.119,E2 -17924.119} C_VEL
LIN {X 0,Y 268.175,Z 445.748,A -85,B 0,C 180,E1 -17926.756,E2 -17926.756} C_VEL
LIN {X 0,Y 268.578,Z 445.465,A -85,B 0,C 180,E1 -17929.606,E2 -17929.606} C_VEL
LIN {X 0,Y 268.996,Z 444.52,A -85,B 0,C 180,E1 -17931.456,E2 -17931.456} C_VEL
LIN {X 0,Y 270.034,Z 441.784,A -85,B 0,C 180,E1 -17934.368,E2 -17934.368} C_VEL
LIN {X 0,Y 271.312,Z 437.988,A -85,B 0,C 180,E1 -17936.957,E2 -17936.957} C_VEL
LIN {X 0,Y 272.883,Z 433.246,A -85,B 0,C 180,E1 -17939.297,E2 -17939.297} C_VEL
LIN {X 0,Y 274.763,Z 427.116,A -85,B 0,C 180,E1 -17941.625,E2 -17941.625} C_VEL
LIN {X 0,Y 277.061,Z 419.38,A -85,B 0,C 180,E1 -17943.921,E2 -17943.921} C_VEL
LIN {X 0,Y 279.176,Z 411.642,A -85,B 0,C 180,E1 -17945.757,E2 -17945.757} C_VEL
LIN {X 0,Y 281.399,Z 402.598,A -85,B 0,C 180,E1 -17947.5,E2 -17947.5} C_VEL
LIN {X 0,Y 283.934,Z 391.738,A -85,B 0,C 180,E1 -17949.136,E2 -17949.136} C_VEL
LIN {X 0,Y 286.04,Z 380.351,A -85,B 0,C 180,E1 -17950.504,E2 -17950.504} C_VEL
LIN {X 0,Y 287.789,Z 368.471,A -85,B 0,C 180,E1 -17951.599,E2 -17951.599} C_VEL
LIN {X 0,Y 289.227,Z 355.65,A -85,B 0,C 180,E1 -17952.458,E2 -17952.458} C_VEL
LIN {X 0,Y 290.18,Z 342.569,A -85,B 0,C 180,E1 -17953.048,E2 -17953.048} C_VEL
LIN {X 0,Y 292.641,Z 278.274,A -85,B 0,C 180,E1 -17954.661,E2 -17954.661} C_VEL
LIN {X 0,Y 286.336,Z 264.618,A -85,B 0,C 180,E1 -17955.974,E2 -17955.974} C_VEL
LIN {X 0,Y 279.02,Z 250.926,A -85,B 0,C 180,E1 -17957.543,E2 -17957.543} C_VEL
LIN {X 0,Y 274.437,Z 243.368,A -85,B 0,C 180,E1 -17958.553,E2 -17958.553} C_VEL
LIN {X 0,Y 272.382,Z 240.08,A -85,B 0,C 180,E1 -17959.018,E2 -17959.018} C_VEL
LIN {X 0,Y 270.725,Z 237.61,A -85,B 0,C 180,E1 -17959.395,E2 -17959.395} C_VEL
LIN {X 0,Y 270.306,Z 236.169,A -85,B 0,C 180,E1 -17959.581,E2 -17959.581} C_VEL
LIN {X 0,Y 270.244,Z 235.818,A -85,B 0,C 180,E1 -17959.937,E2 -17959.937} C_VEL
LIN {X 0,Y 270.245,Z 235.823,A -85,B 0,C 180,E1 -17963.722,E2 -17963.722} C_VEL
LIN {X 0,Y 270.193,Z 235.827,A -85,B 0,C 180,E1 -17966.892,E2 -17966.892} C_VEL
LIN {X 0,Y 270.186,Z 235.825,A -85,B 0,C 180,E1 -17970.382,E2 -17970.382} C_VEL
LIN {X 0,Y 270.252,Z 235.816,A -85,B 0,C 180,E1 -17973.763,E2 -17973.763} C_VEL
LIN {X 0,Y 270.221,Z 235.822,A -85,B 0,C 180,E1 -17977.038,E2 -17977.038} C_VEL
LIN {X 0,Y 270.26,Z 235.812,A -85,B 0,C 180,E1 -17980.854,E2 -17980.854} C_VEL
LIN {X 0,Y 269.576,Z 235.899,A -85,B 0,C 180,E1 -17982.098,E2 -17982.098} C_VEL
LIN {X 0,Y 266.717,Z 236.256,A -85,B 0,C 180,E1 -17984.126,E2 -17984.126} C_VEL
LIN {X 0,Y 264.331,Z 236.557,A -85,B 0,C 180,E1 -17985.776,E2 -17985.776} C_VEL
LIN {X 0,Y 263.351,Z 236.671,A -85,B 0,C 180,E1 -17987.054,E2 -17987.054} C_VEL
LIN {X 0,Y 263.294,Z 236.677,A -85,B 0,C 180,E1 -17987.486,E2 -17987.486} C_VEL
LIN {X 0,Y 263.46,Z 236.661,A -85,B 0,C 180,E1 -17990.79,E2 -17990.79} C_VEL
LIN {X 0,Y 263.49,Z 236.661,A -85,B 0,C 180,E1 -17993.876,E2 -17993.876} C_VEL
LIN {X 0,Y 263.733,Z 236.627,A -85,B 0,C 180,E1 -17998.473,E2 -17998.473} C_VEL
LIN {X 0,Y 263.732,Z 236.617,A -85,B 0,C 180,E1 -18001.527,E2 -18001.527} C_VEL
LIN {X 0,Y 263.514,Z 236.654,A -85,B 0,C 180,E1 -18007.664,E2 -18007.664} C_VEL
LIN {X 0,Y 263.321,Z 236.668,A -85,B 0,C 180,E1 -18010.768,E2 -18010.768} C_VEL
LIN {X 0,Y 263.297,Z 236.675,A -85,B 0,C 180,E1 -18015.482,E2 -18015.482} C_VEL
LIN {X 0,Y 263.197,Z 236.694,A -85,B 0,C 180,E1 -18020.312,E2 -18020.312} C_VEL
LIN {X 0,Y 263.157,Z 236.705,A -85,B 0,C 180,E1 -18025.297,E2 -18025.297} C_VEL
LIN {X 0,Y 263.121,Z 236.708,A -85,B 0,C 180,E1 -18028.737,E2 -18028.737} C_VEL
LIN {X 0,Y 263.112,Z 236.708,A -85,B 0,C 180,E1 -18032.292,E2 -18032.292} C_VEL
LIN {X 0,Y 263.15,Z 236.706,A -85,B 0,C 180,E1 -18035.985,E2 -18035.985} C_VEL
LIN {X 0,Y 263.098,Z 236.708,A -85,B 0,C 180,E1 -18039.875,E2 -18039.875} C_VEL
LIN {X 0,Y 263.099,Z 236.713,A -85,B 0,C 180,E1 -18043.99,E2 -18043.99} C_VEL
LIN {X 0,Y 263.119,Z 236.842,A -85,B 0,C 180,E1 -18047.256,E2 -18047.256} C_VEL
LIN {X 0,Y 265.728,Z 245.746,A -85,B 0,C 180,E1 -18051.28,E2 -18051.28} C_VEL
LIN {X 0,Y 268.129,Z 254.746,A -85,B 0,C 180,E1 -18054.994,E2 -18054.994} C_VEL
LIN {X 0,Y 268.275,Z 255.331,A -85,B 0,C 180,E1 -18055.196,E2 -18055.196} C_VEL
LIN {X 0,Y 270.538,Z 259.788,A -85,B 0,C 180,E1 -18055.748,E2 -18055.748} C_VEL
LIN {X 0,Y 277.325,Z 273.48,A -85,B 0,C 180,E1 -18057.335,E2 -18057.335} C_VEL
LIN {X 0,Y 280.916,Z 281.693,A -85,B 0,C 180,E1 -18058.162,E2 -18058.162} C_VEL
LIN {X 0,Y 284.999,Z 305.035,A -85,B 0,C 180,E1 -18059.493,E2 -18059.493} C_VEL
LIN {X 0,Y 285.777,Z 311.178,A -85,B 0,C 180,E1 -18059.792,E2 -18059.792} C_VEL
LIN {X 0,Y 283.502,Z 365.839,A -85,B 0,C 180,E1 -18061.195,E2 -18061.195} C_VEL
LIN {X 0,Y 282.219,Z 379.388,A -85,B 0,C 180,E1 -18061.812,E2 -18061.812} C_VEL
LIN {X 0,Y 280.38,Z 392.203,A -85,B 0,C 180,E1 -18062.676,E2 -18062.676} C_VEL
LIN {X 0,Y 278.147,Z 403.913,A -85,B 0,C 180,E1 -18063.757,E2 -18063.757} C_VEL
LIN {X 0,Y 275.661,Z 415.214,A -85,B 0,C 180,E1 -18065.123,E2 -18065.123} C_VEL
LIN {X 0,Y 273.122,Z 425.437,A -85,B 0,C 180,E1 -18066.694,E2 -18066.694} C_VEL
LIN {X 0,Y 270.358,Z 435.462,A -85,B 0,C 180,E1 -18068.657,E2 -18068.657} C_VEL
LIN {X 0,Y 267.992,Z 443.921,A -85,B 0,C 180,E1 -18070.751,E2 -18070.751} C_VEL
LIN {X 0,Y 265.797,Z 451.448,A -85,B 0,C 180,E1 -18073.09,E2 -18073.09} C_VEL
LIN {X 0,Y 264.047,Z 457.181,A -85,B 0,C 180,E1 -18075.352,E2 -18075.352} C_VEL
LIN {X 0,Y 262.685,Z 461.729,A -85,B 0,C 180,E1 -18077.639,E2 -18077.639} C_VEL
LIN {X 0,Y 262.107,Z 464.143,A -85,B 0,C 180,E1 -18079.18,E2 -18079.18} C_VEL
LIN {X 0,Y 261.667,Z 466.137,A -85,B 0,C 180,E1 -18080.724,E2 -18080.724} C_VEL
LIN {X 0,Y 261.32,Z 467.724,A -85,B 0,C 180,E1 -18082.27,E2 -18082.27} C_VEL
LIN {X 0,Y 261.126,Z 469.402,A -85,B 0,C 180,E1 -18084.768,E2 -18084.768} C_VEL
LIN {X 0,Y 261.164,Z 469.999,A -85,B 0,C 180,E1 -18086.912,E2 -18086.912} C_VEL
LIN {X 0,Y 261.197,Z 469.979,A -85,B 0,C 180,E1 -18088.456,E2 -18088.456} C_VEL
LIN {X 0,Y 261.253,Z 469.553,A -85,B 0,C 180,E1 -18089.997,E2 -18089.997} C_VEL
LIN {X 0,Y 261.229,Z 468.686,A -85,B 0,C 180,E1 -18091.539,E2 -18091.539} C_VEL
LIN {X 0,Y 261.229,Z 467.417,A -85,B 0,C 180,E1 -18093.081,E2 -18093.081} C_VEL
LIN {X 0,Y 261.203,Z 464.672,A -85,B 0,C 180,E1 -18095.413,E2 -18095.413} C_VEL
LIN {X 0,Y 261.358,Z 460.914,A -85,B 0,C 180,E1 -18097.723,E2 -18097.723} C_VEL
LIN {X 0,Y 261.721,Z 455.984,A -85,B 0,C 180,E1 -18100.049,E2 -18100.049} C_VEL
LIN {X 0,Y 262.38,Z 449.753,A -85,B 0,C 180,E1 -18102.37,E2 -18102.37} C_VEL
LIN {X 0,Y 263.506,Z 441.992,A -85,B 0,C 180,E1 -18104.673,E2 -18104.673} C_VEL
LIN {X 0,Y 264.672,Z 434.017,A -85,B 0,C 180,E1 -18106.582,E2 -18106.582} C_VEL
LIN {X 0,Y 266.083,Z 424.265,A -85,B 0,C 180,E1 -18108.474,E2 -18108.474} C_VEL
LIN {X 0,Y 267.482,Z 413.408,A -85,B 0,C 180,E1 -18110.168,E2 -18110.168} C_VEL
LIN {X 0,Y 268.936,Z 402.913,A -85,B 0,C 180,E1 -18111.455,E2 -18111.455} C_VEL
LIN {X 0,Y 270.302,Z 391.414,A -85,B 0,C 180,E1 -18112.546,E2 -18112.546} C_VEL
LIN {X 0,Y 271.55,Z 377.681,A -85,B 0,C 180,E1 -18113.494,E2 -18113.494} C_VEL
LIN {X 0,Y 272.344,Z 364.628,A -85,B 0,C 180,E1 -18114.077,E2 -18114.077} C_VEL
LIN {X 0,Y 273.792,Z 305.788,A -85,B 0,C 180,E1 -18115.627,E2 -18115.627} C_VEL
LIN {X 0,Y 268.03,Z 259.762,A -85,B 0,C 180,E1 -18117.398,E2 -18117.398} C_VEL
LIN {X 0,Y 267.368,Z 256.963,A -85,B 0,C 180,E1 -18117.569,E2 -18117.569} C_VEL
LIN {X 0,Y 264.902,Z 244.639,A -85,B 0,C 180,E1 -18121.579,E2 -18121.579} C_VEL
LIN {X 0,Y 263.189,Z 236.705,A -85,B 0,C 180,E1 -18124.31,E2 -18124.31} C_VEL
LIN {X 0,Y 263.147,Z 236.71,A -85,B 0,C 180,E1 -18127.892,E2 -18127.892} C_VEL
LIN {X 0,Y 263.107,Z 236.714,A -85,B 0,C 180,E1 -18131.888,E2 -18131.888} C_VEL
LIN {X 0,Y 263.121,Z 236.71,A -85,B 0,C 180,E1 -18136.142,E2 -18136.142} C_VEL
LIN {X 0,Y 263.136,Z 236.707,A -85,B 0,C 180,E1 -18140.132,E2 -18140.132} C_VEL
LIN {X 0,Y 263.155,Z 236.705,A -85,B 0,C 180,E1 -18144.016,E2 -18144.016} C_VEL
LIN {X 0,Y 263.113,Z 236.708,A -85,B 0,C 180,E1 -18148.718,E2 -18148.718} C_VEL
LIN {X 0,Y 263.164,Z 236.702,A -85,B 0,C 180,E1 -18152.999,E2 -18152.999} C_VEL
LIN {X 0,Y 263.161,Z 236.7,A -85,B 0,C 180,E1 -18156.384,E2 -18156.384} C_VEL
LIN {X 0,Y 263.255,Z 236.692,A -85,B 0,C 180,E1 -18159.692,E2 -18159.692} C_VEL
LIN {X 0,Y 263.295,Z 236.686,A -85,B 0,C 180,E1 -18164.518,E2 -18164.518} C_VEL
LIN {X 0,Y 263.334,Z 236.68,A -85,B 0,C 180,E1 -18169.232,E2 -18169.232} C_VEL
LIN {X 0,Y 263.535,Z 236.655,A -85,B 0,C 180,E1 -18172.337,E2 -18172.337} C_VEL
LIN {X 0,Y 263.71,Z 236.618,A -85,B 0,C 180,E1 -18178.472,E2 -18178.472} C_VEL
LIN {X 0,Y 263.709,Z 236.622,A -85,B 0,C 180,E1 -18181.527,E2 -18181.527} C_VEL
LIN {X 0,Y 263.513,Z 236.658,A -85,B 0,C 180,E1 -18187.663,E2 -18187.663} C_VEL
LIN {X 0,Y 263.313,Z 236.682,A -85,B 0,C 180,E1 -18190.768,E2 -18190.768} C_VEL
LIN {X 0,Y 263.273,Z 236.689,A -85,B 0,C 180,E1 -18195.482,E2 -18195.482} C_VEL
LIN {X 0,Y 263.174,Z 236.696,A -85,B 0,C 180,E1 -18200.313,E2 -18200.313} C_VEL
LIN {X 0,Y 263.155,Z 236.701,A -85,B 0,C 180,E1 -18205.296,E2 -18205.296} C_VEL
LIN {X 0,Y 263.122,Z 236.693,A -85,B 0,C 180,E1 -18208.736,E2 -18208.736} C_VEL
LIN {X 0,Y 263.098,Z 236.696,A -85,B 0,C 180,E1 -18212.293,E2 -18212.293} C_VEL
LIN {X 0,Y 263.154,Z 236.705,A -85,B 0,C 180,E1 -18216.766,E2 -18216.766} C_VEL
LIN {X 0,Y 263.099,Z 236.701,A -85,B 0,C 180,E1 -18221.597,E2 -18221.597} C_VEL
LIN {X 0,Y 263.083,Z 236.711,A -85,B 0,C 180,E1 -18226.159,E2 -18226.159} C_VEL
LIN {X 0,Y 263.085,Z 236.712,A -85,B 0,C 180,E1 -18230.132,E2 -18230.132} C_VEL
LIN {X 0,Y 263.144,Z 236.701,A -85,B 0,C 180,E1 -18234.022,E2 -18234.022} C_VEL
LIN {X 0,Y 263.117,Z 236.71,A -85,B 0,C 180,E1 -18237.716,E2 -18237.716} C_VEL
LIN {X 0,Y 263.183,Z 236.701,A -85,B 0,C 180,E1 -18241.79,E2 -18241.79} C_VEL
LIN {X 0,Y 263.19,Z 236.7,A -85,B 0,C 180,E1 -18245.217,E2 -18245.217} C_VEL
LIN {X 0,Y 263.227,Z 236.698,A -85,B 0,C 180,E1 -18249.695,E2 -18249.695} C_VEL
LIN {X 0,Y 263.317,Z 236.689,A -85,B 0,C 180,E1 -18254.524,E2 -18254.524} C_VEL
LIN {X 0,Y 263.345,Z 236.686,A -85,B 0,C 180,E1 -18257.233,E2 -18257.233} C_VEL
LIN {X 0,Y 264.244,Z 239.379,A -85,B 0,C 180,E1 -18257.407,E2 -18257.407} C_VEL
LIN {X 0,Y 269.521,Z 251.876,A -85,B 0,C 180,E1 -18258.235,E2 -18258.235} C_VEL
LIN {X 0,Y 274.845,Z 267.751,A -85,B 0,C 180,E1 -18259.129,E2 -18259.129} C_VEL
LIN {X 0,Y 272.569,Z 342.533,A -85,B 0,C 180,E1 -18261.075,E2 -18261.075} C_VEL
LIN {X 0,Y 271.919,Z 356.02,A -85,B 0,C 180,E1 -18261.737,E2 -18261.737} C_VEL
LIN {X 0,Y 270.979,Z 367.46,A -85,B 0,C 180,E1 -18262.552,E2 -18262.552} C_VEL
LIN {X 0,Y 269.906,Z 378.915,A -85,B 0,C 180,E1 -18263.65,E2 -18263.65} C_VEL
LIN {X 0,Y 268.586,Z 390.662,A -85,B 0,C 180,E1 -18265.125,E2 -18265.125} C_VEL
LIN {X 0,Y 267.139,Z 401.082,A -85,B 0,C 180,E1 -18266.772,E2 -18266.772} C_VEL
LIN {X 0,Y 265.812,Z 409.875,A -85,B 0,C 180,E1 -18268.488,E2 -18268.488} C_VEL
LIN {X 0,Y 264.555,Z 417.841,A -85,B 0,C 180,E1 -18270.383,E2 -18270.383} C_VEL
LIN {X 0,Y 263.404,Z 425.607,A -85,B 0,C 180,E1 -18272.679,E2 -18272.679} C_VEL
LIN {X 0,Y 262.407,Z 432.752,A -85,B 0,C 180,E1 -18275.381,E2 -18275.381} C_VEL
LIN {X 0,Y 261.82,Z 437.51,A -85,B 0,C 180,E1 -18277.715,E2 -18277.715} C_VEL
LIN {X 0,Y 261.356,Z 441.158,A -85,B 0,C 180,E1 -18280.068,E2 -18280.068} C_VEL
LIN {X 0,Y 261.118,Z 443.771,A -85,B 0,C 180,E1 -18282.436,E2 -18282.436} C_VEL
LIN {X 0,Y 261.045,Z 445.113,A -85,B 0,C 180,E1 -18284.257,E2 -18284.257} C_VEL
LIN {X 0,Y 261.122,Z 446.114,A -85,B 0,C 180,E1 -18287.222,E2 -18287.222} C_VEL
LIN {X 0,Y 261.527,Z 445.799,A -85,B 0,C 180,E1 -18289.857,E2 -18289.857} C_VEL
LIN {X 0,Y 262.077,Z 444.649,A -85,B 0,C 180,E1 -18292.052,E2 -18292.052} C_VEL
LIN {X 0,Y 263.085,Z 442.138,A -85,B 0,C 180,E1 -18294.734,E2 -18294.734} C_VEL
LIN {X 0,Y 264.174,Z 439.146,A -85,B 0,C 180,E1 -18296.889,E2 -18296.889} C_VEL
LIN {X 0,Y 265.656,Z 434.901,A -85,B 0,C 180,E1 -18299.189,E2 -18299.189} C_VEL
LIN {X 0,Y 267.666,Z 428.903,A -85,B 0,C 180,E1 -18301.677,E2 -18301.677} C_VEL
LIN {X 0,Y 269.892,Z 421.821,A -85,B 0,C 180,E1 -18303.956,E2 -18303.956} C_VEL
LIN {X 0,Y 272.231,Z 413.932,A -85,B 0,C 180,E1 -18305.966,E2 -18305.966} C_VEL
LIN {X 0,Y 274.712,Z 404.603,A -85,B 0,C 180,E1 -18307.878,E2 -18307.878} C_VEL
LIN {X 0,Y 277.264,Z 394.238,A -85,B 0,C 180,E1 -18309.557,E2 -18309.557} C_VEL
LIN {X 0,Y 279.297,Z 384.159,A -85,B 0,C 180,E1 -18310.861,E2 -18310.861} C_VEL
LIN {X 0,Y 281.218,Z 372.592,A -85,B 0,C 180,E1 -18312.036,E2 -18312.036} C_VEL
LIN {X 0,Y 282.842,Z 360.169,A -85,B 0,C 180,E1 -18312.98,E2 -18312.98} C_VEL
LIN {X 0,Y 283.917,Z 348.125,A -85,B 0,C 180,E1 -18313.629,E2 -18313.629} C_VEL
LIN {X 0,Y 284.695,Z 333.31,A -85,B 0,C 180,E1 -18314.098,E2 -18314.098} C_VEL
LIN {X 0,Y 286.83,Z 280.504,A -85,B 0,C 180,E1 -18315.413,E2 -18315.413} C_VEL
LIN {X 0,Y 280.079,Z 266.071,A -85,B 0,C 180,E1 -18316.883,E2 -18316.883} C_VEL
LIN {X 0,Y 273.099,Z 253.064,A -85,B 0,C 180,E1 -18318.454,E2 -18318.454} C_VEL
LIN {X 0,Y 268.088,Z 245.102,A -85,B 0,C 180,E1 -18319.609,E2 -18319.609} C_VEL
LIN {X 0,Y 265.448,Z 241.069,A -85,B 0,C 180,E1 -18320.242,E2 -18320.242} C_VEL
LIN {X 0,Y 263.721,Z 238.71,A -85,B 0,C 180,E1 -18320.656,E2 -18320.656} C_VEL
LIN {X 0,Y 263.179,Z 236.702,A -85,B 0,C 180,E1 -18320.883,E2 -18320.883} C_VEL
LIN {X 0,Y 263.178,Z 236.702,A -85,B 0,C 180,E1 -18324.021,E2 -18324.021} C_VEL
LIN {X 0,Y 263.123,Z 236.701,A -85,B 0,C 180,E1 -18327.711,E2 -18327.711} C_VEL
LIN {X 0,Y 263.187,Z 236.69,A -85,B 0,C 180,E1 -18331.785,E2 -18331.785} C_VEL
LIN {X 0,Y 263.216,Z 236.685,A -85,B 0,C 180,E1 -18335.2,E2 -18335.2} C_VEL
LIN {X 0,Y 263.252,Z 236.683,A -85,B 0,C 180,E1 -18339.693,E2 -18339.693} C_VEL
LIN {X 0,Y 263.331,Z 236.682,A -85,B 0,C 180,E1 -18344.521,E2 -18344.521} C_VEL
LIN {X 0,Y 263.294,Z 236.677,A -85,B 0,C 180,E1 -18347.486,E2 -18347.486} C_VEL
LIN {X 0,Y 262.718,Z 236.756,A -85,B 0,C 180,E1 -18348.765,E2 -18348.765} C_VEL
LIN {X 0,Y 259.998,Z 237.096,A -85,B 0,C 180,E1 -18350.853,E2 -18350.853} C_VEL
LIN {X 0,Y 256.765,Z 237.497,A -85,B 0,C 180,E1 -18353.42,E2 -18353.42} C_VEL
LIN {X 0,Y 256.382,Z 237.54,A -85,B 0,C 180,E1 -18354.308,E2 -18354.308} C_VEL
LIN {X 0,Y 256.696,Z 237.504,A -85,B 0,C 180,E1 -18358.432,E2 -18358.432} C_VEL
LIN {X 0,Y 256.695,Z 237.493,A -85,B 0,C 180,E1 -18361.569,E2 -18361.569} C_VEL
LIN {X 0,Y 256.444,Z 237.523,A -85,B 0,C 180,E1 -18366.294,E2 -18366.294} C_VEL
LIN {X 0,Y 256.391,Z 237.533,A -85,B 0,C 180,E1 -18369.467,E2 -18369.467} C_VEL
LIN {X 0,Y 256.217,Z 237.556,A -85,B 0,C 180,E1 -18374.293,E2 -18374.293} C_VEL
LIN {X 0,Y 256.141,Z 237.574,A -85,B 0,C 180,E1 -18377.567,E2 -18377.567} C_VEL
LIN {X 0,Y 256.111,Z 237.583,A -85,B 0,C 180,E1 -18381.098,E2 -18381.098} C_VEL
LIN {X 0,Y 256.124,Z 237.583,A -85,B 0,C 180,E1 -18385.112,E2 -18385.112} C_VEL
LIN {X 0,Y 256.043,Z 237.591,A -85,B 0,C 180,E1 -18389.609,E2 -18389.609} C_VEL
LIN {X 0,Y 256.056,Z 237.589,A -85,B 0,C 180,E1 -18393.295,E2 -18393.295} C_VEL
LIN {X 0,Y 256.112,Z 237.577,A -85,B 0,C 180,E1 -18397.272,E2 -18397.272} C_VEL
LIN {X 0,Y 256.045,Z 237.57,A -85,B 0,C 180,E1 -18401.206,E2 -18401.206} C_VEL
LIN {X 0,Y 256.023,Z 237.591,A -85,B 0,C 180,E1 -18405.539,E2 -18405.539} C_VEL
LIN {X 0,Y 256.068,Z 237.707,A -85,B 0,C 180,E1 -18406.024,E2 -18406.024} C_VEL
LIN {X 0,Y 258.604,Z 246.202,A -85,B 0,C 180,E1 -18410.082,E2 -18410.082} C_VEL
LIN {X 0,Y 260.882,Z 254.586,A -85,B 0,C 180,E1 -18413.725,E2 -18413.725} C_VEL
LIN {X 0,Y 262.045,Z 257.23,A -85,B 0,C 180,E1 -18414.11,E2 -18414.11} C_VEL
LIN {X 0,Y 264.186,Z 261.078,A -85,B 0,C 180,E1 -18414.653,E2 -18414.653} C_VEL
LIN {X 0,Y 270.573,Z 273.514,A -85,B 0,C 180,E1 -18416.221,E2 -18416.221} C_VEL
LIN {X 0,Y 275.598,Z 284.914,A -85,B 0,C 180,E1 -18417.433,E2 -18417.433} C_VEL
LIN {X 0,Y 279.586,Z 308.838,A -85,B 0,C 180,E1 -18418.822,E2 -18418.822} C_VEL
LIN {X 0,Y 279.954,Z 312.547,A -85,B 0,C 180,E1 -18418.994,E2 -18418.994} C_VEL
LIN {X 0,Y 277.642,Z 365.618,A -85,B 0,C 180,E1 -18420.381,E2 -18420.381} C_VEL
LIN {X 0,Y 276.304,Z 379.231,A -85,B 0,C 180,E1 -18421.013,E2 -18421.013} C_VEL
LIN {X 0,Y 274.464,Z 391.323,A -85,B 0,C 180,E1 -18421.828,E2 -18421.828} C_VEL
LIN {X 0,Y 272.178,Z 403.156,A -85,B 0,C 180,E1 -18422.928,E2 -18422.928} C_VEL
LIN {X 0,Y 269.599,Z 414.534,A -85,B 0,C 180,E1 -18424.317,E2 -18424.317} C_VEL
LIN {X 0,Y 266.94,Z 424.821,A -85,B 0,C 180,E1 -18425.915,E2 -18425.915} C_VEL
LIN {X 0,Y 264.271,Z 434.099,A -85,B 0,C 180,E1 -18427.73,E2 -18427.73} C_VEL
LIN {X 0,Y 261.532,Z 443.204,A -85,B 0,C 180,E1 -18429.99,E2 -18429.99} C_VEL
LIN {X 0,Y 259.312,Z 450.408,A -85,B 0,C 180,E1 -18432.247,E2 -18432.247} C_VEL
LIN {X 0,Y 257.774,Z 455.377,A -85,B 0,C 180,E1 -18434.177,E2 -18434.177} C_VEL
LIN {X 0,Y 256.132,Z 460.233,A -85,B 0,C 180,E1 -18436.511,E2 -18436.511} C_VEL
LIN {X 0,Y 255.102,Z 463.997,A -85,B 0,C 180,E1 -18438.879,E2 -18438.879} C_VEL
LIN {X 0,Y 254.625,Z 465.961,A -85,B 0,C 180,E1 -18440.466,E2 -18440.466} C_VEL
LIN {X 0,Y 254.261,Z 467.511,A -85,B 0,C 180,E1 -18442.054,E2 -18442.054} C_VEL
LIN {X 0,Y 254.016,Z 469.343,A -85,B 0,C 180,E1 -18445.237,E2 -18445.237} C_VEL
LIN {X 0,Y 254.074,Z 469.684,A -85,B 0,C 180,E1 -18446.826,E2 -18446.826} C_VEL
LIN {X 0,Y 254.122,Z 469.637,A -85,B 0,C 180,E1 -18448.413,E2 -18448.413} C_VEL
LIN {X 0,Y 254.175,Z 469.156,A -85,B 0,C 180,E1 -18449.997,E2 -18449.997} C_VEL
LIN {X 0,Y 254.155,Z 468.261,A -85,B 0,C 180,E1 -18451.582,E2 -18451.582} C_VEL
LIN {X 0,Y 254.138,Z 466.962,A -85,B 0,C 180,E1 -18453.168,E2 -18453.168} C_VEL
LIN {X 0,Y 254.126,Z 464.419,A -85,B 0,C 180,E1 -18455.371,E2 -18455.371} C_VEL
LIN {X 0,Y 254.308,Z 460.336,A -85,B 0,C 180,E1 -18457.939,E2 -18457.939} C_VEL
LIN {X 0,Y 254.691,Z 455.338,A -85,B 0,C 180,E1 -18460.329,E2 -18460.329} C_VEL
LIN {X 0,Y 255.398,Z 449.031,A -85,B 0,C 180,E1 -18462.713,E2 -18462.713} C_VEL
LIN {X 0,Y 256.549,Z 441.137,A -85,B 0,C 180,E1 -18465.08,E2 -18465.08} C_VEL
LIN {X 0,Y 257.729,Z 433.048,A -85,B 0,C 180,E1 -18467.042,E2 -18467.042} C_VEL
LIN {X 0,Y 259.307,Z 423.183,A -85,B 0,C 180,E1 -18468.975,E2 -18468.975} C_VEL
LIN {X 0,Y 260.581,Z 413.476,A -85,B 0,C 180,E1 -18470.52,E2 -18470.52} C_VEL
LIN {X 0,Y 262.075,Z 403.08,A -85,B 0,C 180,E1 -18471.839,E2 -18471.839} C_VEL
LIN {X 0,Y 263.601,Z 390.637,A -85,B 0,C 180,E1 -18473.048,E2 -18473.048} C_VEL
LIN {X 0,Y 264.824,Z 377.513,A -85,B 0,C 180,E1 -18473.972,E2 -18473.972} C_VEL
LIN {X 0,Y 265.637,Z 364.603,A -85,B 0,C 180,E1 -18474.569,E2 -18474.569} C_VEL
LIN {X 0,Y 267.146,Z 306.511,A -85,B 0,C 180,E1 -18476.136,E2 -18476.136} C_VEL
LIN {X 0,Y 261.667,Z 262.297,A -85,B 0,C 180,E1 -18477.887,E2 -18477.887} C_VEL
LIN {X 0,Y 260.091,Z 256.692,A -85,B 0,C 180,E1 -18478.206,E2 -18478.206} C_VEL
LIN {X 0,Y 258.01,Z 246.324,A -85,B 0,C 180,E1 -18481.687,E2 -18481.687} C_VEL
LIN {X 0,Y 256.116,Z 237.585,A -85,B 0,C 180,E1 -18484.819,E2 -18484.819} C_VEL
LIN {X 0,Y 256.107,Z 237.586,A -85,B 0,C 180,E1 -18487.268,E2 -18487.268} C_VEL
LIN {X 0,Y 256.055,Z 237.59,A -85,B 0,C 180,E1 -18492.176,E2 -18492.176} C_VEL
LIN {X 0,Y 256.079,Z 237.585,A -85,B 0,C 180,E1 -18496.676,E2 -18496.676} C_VEL
LIN {X 0,Y 256.085,Z 237.583,A -85,B 0,C 180,E1 -18500.86,E2 -18500.86} C_VEL
LIN {X 0,Y 256.126,Z 237.578,A -85,B 0,C 180,E1 -18502.866,E2 -18502.866} C_VEL
LIN {X 0,Y 256.042,Z 237.588,A -85,B 0,C 180,E1 -18506.703,E2 -18506.703} C_VEL
LIN {X 0,Y 256.086,Z 237.582,A -85,B 0,C 180,E1 -18510.396,E2 -18510.396} C_VEL
LIN {X 0,Y 256.161,Z 237.574,A -85,B 0,C 180,E1 -18514.857,E2 -18514.857} C_VEL
LIN {X 0,Y 256.201,Z 237.572,A -85,B 0,C 180,E1 -18519.107,E2 -18519.107} C_VEL
LIN {X 0,Y 256.231,Z 237.566,A -85,B 0,C 180,E1 -18524.08,E2 -18524.08} C_VEL
LIN {X 0,Y 256.269,Z 237.557,A -85,B 0,C 180,E1 -18528.932,E2 -18528.932} C_VEL
LIN {X 0,Y 256.503,Z 237.531,A -85,B 0,C 180,E1 -18532.125,E2 -18532.125} C_VEL
LIN {X 0,Y 256.674,Z 237.493,A -85,B 0,C 180,E1 -18538.43,E2 -18538.43} C_VEL
LIN {X 0,Y 256.673,Z 237.497,A -85,B 0,C 180,E1 -18541.569,E2 -18541.569} C_VEL
LIN {X 0,Y 256.427,Z 237.538,A -85,B 0,C 180,E1 -18546.802,E2 -18546.802} C_VEL
LIN {X 0,Y 256.367,Z 237.546,A -85,B 0,C 180,E1 -18549.467,E2 -18549.467} C_VEL
LIN {X 0,Y 256.194,Z 237.57,A -85,B 0,C 180,E1 -18554.293,E2 -18554.293} C_VEL
LIN {X 0,Y 256.127,Z 237.576,A -85,B 0,C 180,E1 -18557.567,E2 -18557.567} C_VEL
LIN {X 0,Y 256.088,Z 237.584,A -85,B 0,C 180,E1 -18561.1,E2 -18561.1} C_VEL
LIN {X 0,Y 256.136,Z 237.576,A -85,B 0,C 180,E1 -18565.131,E2 -18565.131} C_VEL
LIN {X 0,Y 256.081,Z 237.57,A -85,B 0,C 180,E1 -18568.587,E2 -18568.587} C_VEL
LIN {X 0,Y 256.043,Z 237.57,A -85,B 0,C 180,E1 -18571.704,E2 -18571.704} C_VEL
LIN {X 0,Y 256.054,Z 237.585,A -85,B 0,C 180,E1 -18575.197,E2 -18575.197} C_VEL
LIN {X 0,Y 256.087,Z 237.583,A -85,B 0,C 180,E1 -18577.274,E2 -18577.274} C_VEL
LIN {X 0,Y 256.029,Z 237.581,A -85,B 0,C 180,E1 -18581.208,E2 -18581.208} C_VEL
LIN {X 0,Y 256.019,Z 237.587,A -85,B 0,C 180,E1 -18585.538,E2 -18585.538} C_VEL
LIN {X 0,Y 256.033,Z 237.591,A -85,B 0,C 180,E1 -18588.801,E2 -18588.801} C_VEL
LIN {X 0,Y 256.111,Z 237.574,A -85,B 0,C 180,E1 -18592.872,E2 -18592.872} C_VEL
LIN {X 0,Y 256.052,Z 237.589,A -85,B 0,C 180,E1 -18596.712,E2 -18596.712} C_VEL
LIN {X 0,Y 256.09,Z 237.581,A -85,B 0,C 180,E1 -18600.403,E2 -18600.403} C_VEL
LIN {X 0,Y 256.159,Z 237.575,A -85,B 0,C 180,E1 -18604.875,E2 -18604.875} C_VEL
LIN {X 0,Y 256.139,Z 237.579,A -85,B 0,C 180,E1 -18609.107,E2 -18609.107} C_VEL
LIN {X 0,Y 256.239,Z 237.572,A -85,B 0,C 180,E1 -18614.085,E2 -18614.085} C_VEL
LIN {X 0,Y 256.269,Z 237.567,A -85,B 0,C 180,E1 -18616.598,E2 -18616.598} C_VEL
LIN {X 0,Y 257.324,Z 240.498,A -85,B 0,C 180,E1 -18616.791,E2 -18616.791} C_VEL
LIN {X 0,Y 263.309,Z 254.498,A -85,B 0,C 180,E1 -18617.765,E2 -18617.765} C_VEL
LIN {X 0,Y 268.154,Z 268.73,A -85,B 0,C 180,E1 -18618.6,E2 -18618.6} C_VEL
LIN {X 0,Y 265.877,Z 342.977,A -85,B 0,C 180,E1 -18620.583,E2 -18620.583} C_VEL
LIN {X 0,Y 265.212,Z 356.094,A -85,B 0,C 180,E1 -18621.239,E2 -18621.239} C_VEL
LIN {X 0,Y 264.193,Z 368.701,A -85,B 0,C 180,E1 -18622.168,E2 -18622.168} C_VEL
LIN {X 0,Y 263.033,Z 379.931,A -85,B 0,C 180,E1 -18623.29,E2 -18623.29} C_VEL
LIN {X 0,Y 261.69,Z 391.522,A -85,B 0,C 180,E1 -18624.803,E2 -18624.803} C_VEL
LIN {X 0,Y 260.195,Z 401.79,A -85,B 0,C 180,E1 -18626.48,E2 -18626.48} C_VEL
LIN {X 0,Y 258.686,Z 411.437,A -85,B 0,C 180,E1 -18628.446,E2 -18628.446} C_VEL
LIN {X 0,Y 257.237,Z 420.527,A -85,B 0,C 180,E1 -18630.785,E2 -18630.785} C_VEL
LIN {X 0,Y 256.106,Z 427.856,A -85,B 0,C 180,E1 -18633.149,E2 -18633.149} C_VEL
LIN {X 0,Y 255.276,Z 433.72,A -85,B 0,C 180,E1 -18635.532,E2 -18635.532} C_VEL
LIN {X 0,Y 254.678,Z 438.337,A -85,B 0,C 180,E1 -18637.933,E2 -18637.933} C_VEL
LIN {X 0,Y 254.211,Z 441.862,A -85,B 0,C 180,E1 -18640.354,E2 -18640.354} C_VEL
LIN {X 0,Y 253.99,Z 444.362,A -85,B 0,C 180,E1 -18642.791,E2 -18642.791} C_VEL
LIN {X 0,Y 253.944,Z 445.47,A -85,B 0,C 180,E1 -18644.424,E2 -18644.424} C_VEL
LIN {X 0,Y 253.929,Z 446.177,A -85,B 0,C 180,E1 -18646.069,E2 -18646.069} C_VEL
LIN {X 0,Y 254.078,Z 446.48,A -85,B 0,C 180,E1 -18647.715,E2 -18647.715} C_VEL
LIN {X 0,Y 254.486,Z 446.133,A -85,B 0,C 180,E1 -18650.124,E2 -18650.124} C_VEL
LIN {X 0,Y 255.197,Z 444.78,A -85,B 0,C 180,E1 -18652.679,E2 -18652.679} C_VEL
LIN {X 0,Y 256.149,Z 442.494,A -85,B 0,C 180,E1 -18655.12,E2 -18655.12} C_VEL
LIN {X 0,Y 257.515,Z 439.03,A -85,B 0,C 180,E1 -18657.643,E2 -18657.643} C_VEL
LIN {X 0,Y 259.317,Z 434.202,A -85,B 0,C 180,E1 -18660.212,E2 -18660.212} C_VEL
LIN {X 0,Y 261.648,Z 427.354,A -85,B 0,C 180,E1 -18662.932,E2 -18662.932} C_VEL
LIN {X 0,Y 264.255,Z 419.475,A -85,B 0,C 180,E1 -18665.341,E2 -18665.341} C_VEL
LIN {X 0,Y 267.035,Z 410.105,A -85,B 0,C 180,E1 -18667.566,E2 -18667.566} C_VEL
LIN {X 0,Y 269.689,Z 400.149,A -85,B 0,C 180,E1 -18669.434,E2 -18669.434} C_VEL
LIN {X 0,Y 272.146,Z 389.993,A -85,B 0,C 180,E1 -18670.937,E2 -18670.937} C_VEL
LIN {X 0,Y 274.327,Z 378.698,A -85,B 0,C 180,E1 -18672.259,E2 -18672.259} C_VEL
LIN {X 0,Y 276.078,Z 367.285,A -85,B 0,C 180,E1 -18673.292,E2 -18673.292} C_VEL
LIN {X 0,Y 277.548,Z 354.612,A -85,B 0,C 180,E1 -18674.133,E2 -18674.133} C_VEL
LIN {X 0,Y 278.448,Z 343.021,A -85,B 0,C 180,E1 -18674.648,E2 -18674.648} C_VEL
LIN {X 0,Y 281.018,Z 282.587,A -85,B 0,C 180,E1 -18676.208,E2 -18676.208} C_VEL
LIN {X 0,Y 274.002,Z 267.731,A -85,B 0,C 180,E1 -18677.811,E2 -18677.811} C_VEL
LIN {X 0,Y 266.66,Z 254.34,A -85,B 0,C 180,E1 -18679.545,E2 -18679.545} C_VEL
LIN {X 0,Y 260.888,Z 245.741,A -85,B 0,C 180,E1 -18680.952,E2 -18680.952} C_VEL
LIN {X 0,Y 258.564,Z 242.081,A -85,B 0,C 180,E1 -18681.554,E2 -18681.554} C_VEL
LIN {X 0,Y 256.841,Z 239.846,A -85,B 0,C 180,E1 -18681.993,E2 -18681.993} C_VEL
LIN {X 0,Y 256.145,Z 237.573,A -85,B 0,C 180,E1 -18682.278,E2 -18682.278} C_VEL
LIN {X 0,Y 256.068,Z 237.587,A -85,B 0,C 180,E1 -18686.708,E2 -18686.708} C_VEL
LIN {X 0,Y 256.095,Z 237.58,A -85,B 0,C 180,E1 -18690.398,E2 -18690.398} C_VEL
LIN {X 0,Y 256.178,Z 237.561,A -85,B 0,C 180,E1 -18694.862,E2 -18694.862} C_VEL
LIN {X 0,Y 256.155,Z 237.564,A -85,B 0,C 180,E1 -18699.104,E2 -18699.104} C_VEL
LIN {X 0,Y 256.267,Z 237.556,A -85,B 0,C 180,E1 -18704.083,E2 -18704.083} C_VEL
LIN {X 0,Y 256.278,Z 237.559,A -85,B 0,C 180,E1 -18708.933,E2 -18708.933} C_VEL
LIN {X 0,Y 256.497,Z 237.521,A -85,B 0,C 180,E1 -18712.126,E2 -18712.126} C_VEL
LIN {X 0,Y 256.382,Z 237.54,A -85,B 0,C 180,E1 -18714.308,E2 -18714.308} C_VEL
LIN {X 0,Y 255.654,Z 237.629,A -85,B 0,C 180,E1 -18715.621,E2 -18715.621} C_VEL
LIN {X 0,Y 252.918,Z 237.97,A -85,B 0,C 180,E1 -18717.769,E2 -18717.769} C_VEL
LIN {X 0,Y 250.663,Z 238.253,A -85,B 0,C 180,E1 -18719.516,E2 -18719.516} C_VEL
LIN {X 0,Y 249.719,Z 238.362,A -85,B 0,C 180,E1 -18720.865,E2 -18720.865} C_VEL
LIN {X 0,Y 249.65,Z 238.369,A -85,B 0,C 180,E1 -18721.322,E2 -18721.322} C_VEL
LIN {X 0,Y 249.415,Z 238.4,A -85,B 0,C 180,E1 -18726.472,E2 -18726.472} C_VEL
LIN {X 0,Y 249.323,Z 238.411,A -85,B 0,C 180,E1 -18729.738,E2 -18729.738} C_VEL
LIN {X 0,Y 249.158,Z 238.433,A -85,B 0,C 180,E1 -18734.707,E2 -18734.707} C_VEL
LIN {X 0,Y 249.072,Z 238.452,A -85,B 0,C 180,E1 -18738.083,E2 -18738.083} C_VEL
LIN {X 0,Y 249.036,Z 238.463,A -85,B 0,C 180,E1 -18741.523,E2 -18741.523} C_VEL
LIN {X 0,Y 249.075,Z 238.459,A -85,B 0,C 180,E1 -18745.459,E2 -18745.459} C_VEL
LIN {X 0,Y 249.026,Z 238.466,A -85,B 0,C 180,E1 -18748.973,E2 -18748.973} C_VEL
LIN {X 0,Y 248.992,Z 238.468,A -85,B 0,C 180,E1 -18752.432,E2 -18752.432} C_VEL
LIN {X 0,Y 249.01,Z 238.468,A -85,B 0,C 180,E1 -18756.349,E2 -18756.349} C_VEL
LIN {X 0,Y 248.986,Z 238.455,A -85,B 0,C 180,E1 -18760.483,E2 -18760.483} C_VEL
LIN {X 0,Y 249.03,Z 238.657,A -85,B 0,C 180,E1 -18764.732,E2 -18764.732} C_VEL
LIN {X 0,Y 251.562,Z 247.038,A -85,B 0,C 180,E1 -18768.966,E2 -18768.966} C_VEL
LIN {X 0,Y 253.667,Z 254.44,A -85,B 0,C 180,E1 -18772.317,E2 -18772.317} C_VEL
LIN {X 0,Y 256.25,Z 259.138,A -85,B 0,C 180,E1 -18773.033,E2 -18773.033} C_VEL
LIN {X 0,Y 261.996,Z 270.039,A -85,B 0,C 180,E1 -18774.563,E2 -18774.563} C_VEL
LIN {X 0,Y 267.694,Z 281.885,A -85,B 0,C 180,E1 -18776.011,E2 -18776.011} C_VEL
LIN {X 0,Y 270.356,Z 288.181,A -85,B 0,C 180,E1 -18776.681,E2 -18776.681} C_VEL
LIN {X 0,Y 274.017,Z 311.186,A -85,B 0,C 180,E1 -18778.042,E2 -18778.042} C_VEL
LIN {X 0,Y 274.112,Z 314.788,A -85,B 0,C 180,E1 -18778.174,E2 -18778.174} C_VEL
LIN {X 0,Y 271.854,Z 365.149,A -85,B 0,C 180,E1 -18779.519,E2 -18779.519} C_VEL
LIN {X 0,Y 270.391,Z 379.001,A -85,B 0,C 180,E1 -18780.164,E2 -18780.164} C_VEL
LIN {X 0,Y 268.469,Z 391.47,A -85,B 0,C 180,E1 -18781.034,E2 -18781.034} C_VEL
LIN {X 0,Y 265.912,Z 403.972,A -85,B 0,C 180,E1 -18782.236,E2 -18782.236} C_VEL
LIN {X 0,Y 263.26,Z 415.14,A -85,B 0,C 180,E1 -18783.652,E2 -18783.652} C_VEL
LIN {X 0,Y 260.499,Z 425.237,A -85,B 0,C 180,E1 -18785.28,E2 -18785.28} C_VEL
LIN {X 0,Y 257.722,Z 434.36,A -85,B 0,C 180,E1 -18787.132,E2 -18787.132} C_VEL
LIN {X 0,Y 255.329,Z 441.921,A -85,B 0,C 180,E1 -18789.032,E2 -18789.032} C_VEL
LIN {X 0,Y 252.936,Z 449.365,A -85,B 0,C 180,E1 -18791.364,E2 -18791.364} C_VEL
LIN {X 0,Y 250.931,Z 455.377,A -85,B 0,C 180,E1 -18793.734,E2 -18793.734} C_VEL
LIN {X 0,Y 249.204,Z 460.162,A -85,B 0,C 180,E1 -18796.129,E2 -18796.129} C_VEL
LIN {X 0,Y 248.114,Z 463.861,A -85,B 0,C 180,E1 -18798.562,E2 -18798.562} C_VEL
LIN {X 0,Y 247.599,Z 465.792,A -85,B 0,C 180,E1 -18800.192,E2 -18800.192} C_VEL
LIN {X 0,Y 247.202,Z 467.286,A -85,B 0,C 180,E1 -18801.826,E2 -18801.826} C_VEL
LIN {X 0,Y 246.925,Z 469.056,A -85,B 0,C 180,E1 -18805.099,E2 -18805.099} C_VEL
LIN {X 0,Y 246.986,Z 469.37,A -85,B 0,C 180,E1 -18806.735,E2 -18806.735} C_VEL
LIN {X 0,Y 247.049,Z 469.282,A -85,B 0,C 180,E1 -18808.367,E2 -18808.367} C_VEL
LIN {X 0,Y 247.098,Z 468.76,A -85,B 0,C 180,E1 -18809.997,E2 -18809.997} C_VEL
LIN {X 0,Y 247.081,Z 467.837,A -85,B 0,C 180,E1 -18811.627,E2 -18811.627} C_VEL
LIN {X 0,Y 247.05,Z 466.508,A -85,B 0,C 180,E1 -18813.258,E2 -18813.258} C_VEL
LIN {X 0,Y 247.027,Z 464.238,A -85,B 0,C 180,E1 -18815.273,E2 -18815.273} C_VEL
LIN {X 0,Y 247.252,Z 459.759,A -85,B 0,C 180,E1 -18818.167,E2 -18818.167} C_VEL
LIN {X 0,Y 247.68,Z 454.692,A -85,B 0,C 180,E1 -18820.625,E2 -18820.625} C_VEL
LIN {X 0,Y 248.438,Z 448.304,A -85,B 0,C 180,E1 -18823.076,E2 -18823.076} C_VEL
LIN {X 0,Y 249.639,Z 440.281,A -85,B 0,C 180,E1 -18825.508,E2 -18825.508} C_VEL
LIN {X 0,Y 250.731,Z 433.028,A -85,B 0,C 180,E1 -18827.312,E2 -18827.312} C_VEL
LIN {X 0,Y 252.361,Z 423.282,A -85,B 0,C 180,E1 -18829.286,E2 -18829.286} C_VEL
LIN {X 0,Y 253.946,Z 412.225,A -85,B 0,C 180,E1 -18831.082,E2 -18831.082} C_VEL
